// TwinCAT 3 PLC project SlaveController
// ProgramVersion: 3.1.4024.0
// libraries:
//   Tc2_Math, * (Beckhoff Automation GmbH)
//   Tc2_Standard, * (Beckhoff Automation GmbH)
//   Tc2_System, * (Beckhoff Automation GmbH)
//   Tc2_Utilities, * (Beckhoff Automation GmbH)
//   Tc3_Module, * (Beckhoff Automation GmbH)
// project tree:
//   AgiMaths/ deg2rad.TcPOU, sign.TcPOU (not stored), addVec7.TcPOU (not stored), atan2.TcPOU (not stored), cot.TcPOU (not stored)
//   AgiMaths/Frames/ DHTrans.TcPOU (not stored), rotX.TcPOU (not stored), rotY.TcPOU (not stored), rotZ.TcPOU (not stored), transform.TcPOU (not stored)
//   AgiMaths/MatrixLib/ cross.TcPOU (not stored), Det5.TcPOU (not stored), Det6.TcPOU (not stored), Det7.TcPOU (not stored), invMat6.TcPOU, invMat6Old.TcPOU (not stored), invMat3.TcPOU (not stored), invMat7.TcPOU (not stored), Mat3T.TcPOU (not stored), matAdd.TcPOU (not stored), matMultiNum.TcPOU (not stored), matMultiply.TcPOU (not stored), matMultiVec.TcPOU (not stored), matSelfAdd.TcPOU (not stored), matSelfSub.TcPOU (not stored), matSub.TcPOU (not stored), matTranspose.TcPOU (not stored), rot2AngAxis.TcPOU (not stored), vecAdd.TcPOU (not stored), vecNorm.TcPOU (not stored), normVec.TcPOU (not stored), vecSelfMultiNum.TcPOU (not stored), vecMultiNum.TcPOU (not stored), vecSub.TcPOU (not stored)
//   DUTs/Enum/ E_SetupArmState.TcDUT, E_DriverCtrlWord.TcDUT (not stored), E_DriverOPMode.TcDUT (not stored), E_DriverStatusWord.TcDUT (not stored)
//   DUTs/Structure/MasterSlaveCommunication/ E_InstrumentType.TcDUT (not stored), E_MasterArmState.TcDUT (not stored), E_MatchedMasterArmIdx.TcDUT (not stored), E_MatchedSlaveArmIdx.TcDUT (not stored), E_SlaveArmState.TcDUT, ST_InstruStatus.TcDUT (not stored), ST_MasterStatus.TcDUT (not stored), ST_SlaveStatus.TcDUT (not stored)
//   DUTs/Structure/ ST_SetupArmCtrlCmds.TcDUT (not stored), ST_SetupInputDataPool.TcDUT (not stored), ST_SlaveArmCtrlCmds.TcDUT, ST_SlaveInputDataPool.TcDUT, ST_InstruParameters.TcDUT, ST_Frame.TcDUT (not stored)
//   DUTs/Structure/TasksCommunication/ ST_SetupStatus.TcDUT, ST_SetupJointData.TcDUT (not stored), ST_SlaveDynaData.TcDUT (not stored), ST_SlaveUIData.TcDUT, ST_CartStatus.TcDUT (not stored), ST_MasterJointData.TcDUT (not stored), ST_MotorInputs.TcDUT (not stored), ST_MotorOutputs.TcDUT (not stored), ST_SlaveJointData.TcDUT, ST_SafetyData.TcDUT (not stored)
//   DUTs/Type/ Mat34.TcDUT (not stored), Mat37.TcDUT (not stored), Mat43.TcDUT (not stored), Mat4d.TcDUT (not stored), Mat5d.TcDUT (not stored), Mat67.TcDUT (not stored), Mat6d.TcDUT (not stored), Mat76.TcDUT (not stored), Mat7d.TcDUT (not stored), Vec4d.TcDUT (not stored), Vec4i.TcDUT (not stored), Vec5d.TcDUT (not stored), Vec5i.TcDUT (not stored), Vec6i.TcDUT (not stored), Vec8d.TcDUT (not stored), Vec8i.TcDUT (not stored), Mat3d.TcDUT (not stored), Vec3d.TcDUT (not stored), Vec6d.TcDUT (not stored), Vec7d.TcDUT (not stored), Vec7i.TcDUT (not stored)
//   FBs_BasicControllers/ FBGripControl.TcPOU (not stored), FBMacroJntControl.TcPOU, FB_PID.TcPOU (not stored)
//   FBs_RobotDynamics/ FB_SlaveGravity.TcPOU, FB_setupSlaveGravity.TcPOU (not stored)
//   FBs_Robots/ FB_Instrument.TcPOU, FB_SetupArm.TcPOU, FB_SlaveJoint.TcPOU, FB_SetupJoint.TcPOU, FB_SetupRobot.TcPOU, FB_JointBase.TcPOU, FB_SlaveArm.TcPOU, FB_SlaveRobot.TcPOU
//   FBs_SetupControllers/ FB_SetupCtrlManualAdjust.TcPOU (not stored), FB_SetupCtrlHold.TcPOU, FB_SetupArmCtrlBase.TcPOU (not stored), FB_SetupCtrlAutoAdjust.TcPOU (not stored), FB_SetupCtrlCart.TcPOU, FB_SetupCtrlError.TcPOU (not stored), FB_SetupCtrlGraCali.TcPOU, FB_SetupCtrlInit.TcPOU (not stored), FB_SetupCtrlPackage.TcPOU, FB_SetupCtrlSelfCheck.TcPOU, I_SetupArmCtrl.TcIO
//   FBs_SlaveControllers/ FB_SlaveCtrlPackage.TcPOU (not stored), FB_SlaveCtrlEndoscope.TcPOU, FB_SlaveCtrlCart.TcPOU (not stored), FB_SlaveCtrlScopeReady.TcPOU, FB_SlaveCtrlSelfCheck.TcPOU, FB_SlaveCtrlError.TcPOU (not stored), FB_SlaveCtrlInstruReady.TcPOU (not stored), FB_SlaveCtrlMasterSlave.TcPOU, FB_SlaveCtrlMountInstru.TcPOU, FB_SlaveCtrlAdjust.TcPOU, FB_SlaveCtrlMountPanel.TcPOU, FB_SlaveCtrlPanelReady.TcPOU (not stored), FB_SlaveCtrlMountScope.TcPOU (not stored), FB_SlaveCtrlGraCali.TcPOU, FB_SlaveCtrlInit.TcPOU (not stored), FB_SlaveCtrlStandBy.TcPOU, FB_SlaveArmCtrlBase.TcPOU, I_SlaveArmCtrl.TcIO (not stored)
//   FBs_TrajectoryPlanning/ FB_BasicDoubleS.TcPOU (not stored), FB_trajBase.TcPOU (not stored), FB_TrajMoveJ.TcPOU, FB_setupTrajMoveJ.TcPOU, linear_trajectory_with_quintic_polynomial_blends.TcPOU (not stored), quintic_spline_curve.TcPOU (not stored), Quintic_spline_curve_factor.TcPOU (not stored), TrapezoIDal_velocity_trajectory.TcPOU (not stored)
//   FBs_TrajectoryPlanning/OTG/ FB_secOrdTrajFilter.TcPOU (not stored), FB_thirdOrdTrajFilter.TcPOU (not stored)
//   FBs_Filters/ FB_LowPassFilter.TcPOU (not stored)
//   GVLs/ GVL_CartParameters.TcGVL (not stored), GVL_InstruCtrlParams.TcGVL, GVL_MathDefine.TcGVL, GVL_SafetyParameters.TcGVL (not stored), GVL_SystemParameters.TcGVL
//   GVLs/SetupArms/ GVL_SetupJointEncoderCaliData.TcGVL, GVL_SetupMotorParameters.TcGVL, GVL_SetupArmKinematic.TcGVL, GVL_SetupControlParameters.TcGVL (not stored)
//   GVLs/SlaveArms/ GVLs_SlaveArmDynamics.TcGVL, GVLs_SetupSlaveArmDynamics.TcGVL, GVL_SlaveArmKinematic.TcGVL, GVL_SlaveControlParameters.TcGVL, GVL_SlaveMotorParameters.TcGVL, GVL_SlaveJointEncoderCaliData.TcGVL
//   Mains/ SetupArmControl.TcPOU (not stored), SlaveArmControl.TcPOU, RobotDynamics.TcPOU
//   / TaskDynamic.TcTTO (not stored), TaskSetupArmControl.TcTTO, TaskSlaveArmControl.TcTTO
// real-time tasks:
//   TASK TaskSlaveArmControl: cycle T#250us, priority 1, ADS port 350
//   TASK TaskDynamic: cycle T#1ms, priority 2, ADS port 351
//   TASK TaskSetupArmControl: cycle T#1ms, priority 3, ADS port 352

CONFIGURATION SlaveController
    RESOURCE PLC ON TwinCAT3
        TASK TaskSetupArmControl(INTERVAL := T#1ms, PRIORITY := 3);
        TASK TaskSlaveArmControl(INTERVAL := T#250us, PRIORITY := 1);
        PROGRAM SetupArmControl WITH TaskSetupArmControl : SetupArmControl;
        PROGRAM SlaveArmControl WITH TaskSlaveArmControl : SlaveArmControl;
    END_RESOURCE
END_CONFIGURATION

// ---- DUTs/Enum/E_SetupArmState.TcDUT
TYPE E_SetupArmState :
(
	SetupArmState_Error := 1,
	SetupArmState_Init :=2,
	SetupArmState_SelfCheck :=3,
	SetupArmState_Hold :=4,
	SetupArmState_ManulAdjust :=5,
	SetupArmState_AutoAdjust :=6,
	SetupArmState_Package :=7,
	SetupArmState_Cart := 8,
	SetupArmState_GravityCali := 9,
	
	SetupArmState_totalNum :=SetupArmState_GravityCali
);
END_TYPE

// ---- DUTs/Structure/MasterSlaveCommunication/E_SlaveArmState.TcDUT
TYPE E_SlaveArmState :
(
	SlaveArmState_Error := 1,
	SlaveArmState_Init :=2,
	SlaveArmState_SelfCheck :=3,
	SlaveArmState_Standby :=4,
	SlaveArmState_MountPanel:=5,
	SlaveArmState_PanelReady :=6,
	SlaveArmState_MountInstru :=7,
	SlaveArmState_InstruReady :=8,
	SlaveArmState_MasterSlave :=9,
	SlaveArmState_MountScope :=10,
	SlaveArmState_ScopeReady :=11,
	SlaveArmState_EndoScope :=12,
	SlaveArmState_Adjust :=13,	
	SlaveArmState_Package :=14,  		 //包装
	SlaveArmState_Cart := 15,    			 //搬运
	SlaveArmState_GravityCali := 16, 	 //重力标定
	
	SlaveArmState_totalNum :=SlaveArmState_GravityCali
);
END_TYPE

// ---- DUTs/Structure/TasksCommunication/ST_SetupStatus.TcDUT
TYPE ST_SetupStatus :
STRUCT
	// state machine
	m_armState:ARRAY[1..g_sArmNum] OF E_SetupArmState:=[g_sArmNum(SetupArmState_Init)];
	
	// current pose of set arm distal end
	m_curEndPose:ARRAY[1..g_sArmNum] OF ST_Frame;
	
	// position of remote center point
	m_rcPos :ARRAY[1..g_sArmNum] OF Vec3d;
END_STRUCT
END_TYPE

// ---- DUTs/Structure/TasksCommunication/ST_SlaveUIData.TcDUT
// Output from UI controller
// Input to slave arm control task and cart control task  
TYPE ST_SlaveUIData :
STRUCT
	m_slaveArmDisableFlag :Vec4i:=[0, 0, 0, 0];
END_STRUCT
END_TYPE

// ---- DUTs/Structure/TasksCommunication/ST_SlaveJointData.TcDUT
TYPE ST_SlaveJointData :
STRUCT
	
	// joint position compute with motor encoder
	m_curMotorPos :ARRAY[1..g_sArmNum] OF Vec8d;
	
	// joint position compute with link/abs encoder
	m_curLinkPos :ARRAY[1..g_sArmNum] OF Vec8d;
	
	// target joint position 
	m_cmdJntPos :ARRAY[1..g_sArmNum] OF Vec8d;
	
	// current joint position 
	m_curJntPos :ARRAY[1..g_sArmNum] OF Vec8d;
	
	// target joint velocity 
	m_cmdJntVel :ARRAY[1..g_sArmNum] OF Vec8d;
	
	// current joint position 
	m_curJntVel :ARRAY[1..g_sArmNum] OF Vec8d;
	
	// command joint torque 
	m_cmdJntTrq :ARRAY[1..g_sArmNum] OF Vec8d;
	
	// current joint torque 
	m_curJntTrq :ARRAY[1..g_sArmNum] OF Vec8d;
	
	// raw joint current  
	m_rawJntCurrent :ARRAY[1..g_sArmNum] OF Vec8d;
	
	// filtd  joint current  
	m_filtJntCurrent :ARRAY[1..g_sArmNum] OF Vec8d;
	
	// command joint current 
	m_cmdJntCurrent :ARRAY[1..g_sArmNum] OF Vec8d;
END_STRUCT
END_TYPE

// ---- DUTs/Structure/ST_SlaveArmCtrlCmds.TcDUT
TYPE ST_SlaveArmCtrlCmds :
STRUCT
	// arm control data
	m_jntEnableFlag : Vec8i;
	m_jntOPMode : Vec8i;
	m_cmdJntPos : VEC8d;
	m_cmdJntVel : VEC8d;
	m_cmdJntAcc : VEC8d;
	m_cmdJntTrq : VEC8d;
	m_cmdCartPose : ST_Frame;
	m_cmdCartTwist : Vec6d;
	m_ratedCur : VEC8d;
	
END_STRUCT
END_TYPE

// ---- DUTs/Structure/ST_SlaveInputDataPool.TcDUT
// Struct contains all data from other tasks and controller used for slave control
TYPE ST_SlaveInputDataPool :
STRUCT
		
	// UI information, import from UI controller
	m_UIData AT %I*:ST_SlaveUIData;
	
	// safety information, import from safety check task
	m_safetyData AT %I*: ST_SafetyData;
	
	// cart information, import from other task
	m_cartStatus AT %I*:ST_CartStatus;
	
	// master robot information, import from other device
	m_masterStatus AT %I*:ST_MasterStatus;
	
	// setup arms infromation;
	m_setupArmStates AT %i* : ST_SetupArmStatus;
	
	// slave dynamic data
	m_slaveDynaData AT %I* : ST_SlaveDynaData;
	
END_STRUCT
END_TYPE

// ---- DUTs/Structure/ST_InstruParameters.TcDUT
 // instrumetn kinematic paramters
TYPE ST_InstruParameters :
STRUCT	
		
	m_rodLength:LREAL:=0.5392; //器械杆长
	m_headLength:LREAL :=0.01;
	m_fingerLenght:LREAL :=0;//器械头端长度 
	
	kx:lreal:=1;
	ky:lreal:=1;
	kz:lreal:=1;

	k13:LREAL:=0.775;
	k23:LREAL:=0.775;
	m_openAngleDir:INT:=-1;

	Len_fixed_point:LREAL:=0.2;	//不动点距离安装面的长度
	Len_mounting_surface:LREAL:=0.009; //器械安装面距离滑块的长度(图中的L3)
	Len_Hight:lreal:=0; //器械杆的高度
	slope_angle:LREAL:=0; //如果器械是摄像头，还需要考虑摄像头的斜面角度
	open_angle_max:LREAL:=1.57;

END_STRUCT
END_TYPE

// ---- GVLs/GVL_InstruCtrlParams.TcGVL
// TODO： Code review and refined
VAR_GLOBAL
	
	//器械相关
	Head_Len_1:ARRAY[1..30] OF LREAL:=[1,1,1,1,1,1,	0.01950, 0.0096, 0.0109, 0.011,		0.01101, 0.02313, 0.0195, 0.0207, 0.0130, 0.01638, 0.01638, 13(1)	];
	
	camera_slope_angle:LREAL:=30.0*g_deg2Rad;; //摄像头斜面角度
	
	a3:ARRAY[1..30] OF LREAL:=[1,1,1,1,1,1,  0.0089,0.0089,0.010,0.010,		0.0089,0.01065,0.01065,0.01065,0.0089,		0.00935,0.00935,0,0,   4(0), 0.0089, 5(0)];
	k13:ARRAY[1..30] OF LREAL:=[1,1,1,1,1,1, 0.77510204, 0.808510638, 0.62295082, 0.644067797,  0.729166667,  0.5, 0.62295082, 0.62295082,  0.729166667,   -0.734693878,	-0.734693878,    1,      1,   1,	4(1), 0.77510204, 5(1)];
	k23:ARRAY[1..30] OF LREAL:=[1,1,1,1,1,1, 0.77510204, 0.808510638, 0.62295082, 0.644067797,  0.729166667,  0.5, 0.62295082, 0.62295082,  0.729166667,   -0.734693878,	-0.734693878,    1,      1,   1,	4(1), 0.77510204, 5(1)  ];
	kx:ARRAY[1..30] OF LREAL:=[30(-1)];
	ky:ARRAY[1..30] OF LREAL:=[1,1,1,1,1,1,  0.931034483,    0.931034483,      0.931034483,    0.931034483,    0.947368421,    0.931034483,    0.931034483,     0.931034483,     0.931034483,   0.877192982,	0.877192982,    1,      1,   1,	4(1), 0.931034483, 5(1)   ];
	kz:ARRAY[1..30] OF LREAL:=[1,1,1,1,1,1,  0.844827586,    0.810344828,      1.051724138,    1.017241379,    0.842105263,    1.310344828,    1.051724138,     1.051724138,     0.827586207,   0.859649123,	0.859649123,    1,      1,   1,	4(1), 0.844827586, 5(1)  ];
	openAngleDir:ARRAY[1..30] OF INT:=[30(-1)];
	
	rad_30:LREAL:=30.0*g_deg2Rad;  rad_60:LREAL:=60.0*g_deg2Rad;	 rad_38:LREAL:=38.0*g_deg2Rad;	rad_55:LREAL:=55.0*g_deg2Rad;	
	rad_45:LREAL:=45.0*g_deg2Rad; rad_28:LREAL:=28.0*g_deg2Rad; rad_10:LREAL:=10.0*g_deg2Rad;rad_90:LREAL:=90.0*g_deg2Rad;
	open_angle_max:ARRAY[1..30] OF LREAL:=[1,1,1,1,1,1,  rad_45,  rad_30+rad_10,  rad_38+rad_10, rad_38+rad_10,	 rad_30+rad_10, rad_90, rad_45+rad_10, rad_45+rad_10,  rad_60,rad_30,     rad_30,1,1];
	
	tool_name:ARRAY[1..30] OF STRING:=['1','1','1','1','1','1',  'Cadiere Forceps','Large Needle Driver','Mega SutureCut Needle Driver','Large SutureCut Needle Driver',	'RoundTip Scissors','Prograsp',	'Maryland Bipolar Forceps','Fenestrated Bipolar Forceps', 'Monopolar Curved Scissors','Permanent Cautery Hook','Permanent Cautery Spatula','1','1','Camera'];
	
//	Head_Len:ARRAY[1..30] OF LREAL:=[1,1,1,1,1,1,	0.01950, 0.0096, 0.0109, 0.011,		0.01101, 0.02313, 0.0195, 0.0207, 0.0130, 0.01638, 0.01638, 13(1)	];
	Head_Len:ARRAY[1..30] OF LREAL:=[0,0,0,0,0,0,	0, 0.0096, 0.0109,  0.0109,		0, 0, 0, 0, 0, 0, 0, 13(0)	];
		
	//*************************绝对定位精度测试使用*****************************//
	len1:LREAL:=0.5438;  len3:LREAL:=0.009;	len_camera:LREAL:=0.49;//0.477;//0.3035;//0.51	
	Len_Rod:ARRAY[1..30] OF LREAL:=[0,0,0,0,0,  0, len1,len1,len1,len1,	len1,len1,len1,len1,0.54375,	0.5432, 0.5432,0,0,len_camera,     4(0),0.551,5(0)]; //器械的杆长	，ID25号器械是主从延时测试用，长度为533+18
	
	Len_mounting_surface:ARRAY[1..30] OF LREAL:=[0,0,0,0,0,	0,len3,len3,len3,len3,	len3,len3,len3,len3,len3,	len3,len3,0,0,len3,    4(0),len3,5(0)]; //滑块和器械安装面的距离(图中的L3)
	TroCar_Len:LREAL:=0.1;//穿刺器长度、此处使用的是短穿刺器
	Zero_To_Bottom_J8:LREAL:=0.14;//8关节刻度线到最底部长度

	
	// Add by NiFeijian,  new method to mount panel and instrument, can be repalced later
	// joint position of panel locked position
	g_panelLockedPosition :Vec5d:=[0.0, 0.0, 0.0, 0.0, 0.0];	
	
	// motor position when instrument is at zero position
	g_instruZeroPosition :Vec5d :=[0.0, 0.0, 0.0, 0.0, 0.0];// move to instrument chip and read online

END_VAR

// ---- GVLs/GVL_MathDefine.TcGVL
VAR_GLOBAL CONSTANT
	g_smallNum :LREAL := 1E-6;
	g_smallAng :LREAL := 0.01*PI/180;
	g_largeNum: LREAL :=1E16;
	g_deg2Rad :LREAL := pi/180.0;
	g_rad2Deg :LREAL := 180.0/pi;
	
	g_eye3d :Mat3d:=[1, 0, 0,
					 0, 1, 0,
					 0, 0, 1];
	g_eye4d :Mat4d:=[1, 0, 0, 0,
					 0, 1, 0, 0,
					 0, 0, 1, 0,
					 0, 0, 0, 1];
	g_zeorMat3d :Mat3d:=[9(0)];
	
	g_zeroMat6d :Mat6d:=[36(0)];
	g_zeroMat7d :Mat7d:=[49(0)];
	g_eye7d :Mat7d:=[1, 0, 0, 0, 0, 0, 0, 
					 0, 1, 0, 0, 0, 0, 0, 
					 0, 0, 1, 0, 0, 0, 0, 
					 0, 0, 0, 1, 0, 0, 0,
					 0, 0, 0, 0, 1, 0, 0,
					 0, 0, 0, 0, 0, 1, 0,
					 0, 0, 0, 0, 0, 0, 1];
	
	g_zeroVec3d :Vec3d:= [3(0)];
	g_onesVec3d: Vec3d:=[3(1)];
	
	g_zeroVec6d: Vec6d:=[6(0)];
	g_onesVec6d: Vec6d:=[6(1)];
	
	g_zeroVec5d: Vec5d:=[5(0)];
	g_onesVec5d: Vec5d:=[5(1.0)];
	g_zeroVec5i: Vec5i:=[5(0)];
	g_onesVec5i: Vec5i:=[5(1)];
	
	g_zeroVec7d: Vec7d:=[7(0)];
	g_onesVec7d: Vec7d:=[7(1.0)];
	g_zeroVec7i: Vec7i:=[7(0)];
	g_onesVec7i: Vec7i:=[7(1)];
	g_zeroVec8d: Vec8d:=[8(0)];
	g_onesVec8d: Vec8d:=[8(1.0)];
	g_zeroVec8i: Vec8i:=[8(0)];
	g_onesVec8i: Vec8i:=[8(1)];
	
	g_setupAllPosMode:Vec5i:=[5(DriverOPMode_Pos)];
	g_setupAllTrqMode:Vec5i:=[5(DriverOPMode_Trq)];
	g_slaveAllPosMode:Vec8i:=[8(DriverOPMode_Pos)];
	g_slaveAllTrqMode:Vec8i:=[8(DriverOPMode_Trq)];
	g_slaveAllPosTrqMode:Vec8i:=[8(DriverOPMode_PosTrq)];
	
	
END_VAR

// ---- GVLs/GVL_SystemParameters.TcGVL
VAR_GLOBAL CONSTANT
	
	g_mArmNum :INT := 2;	
	g_mJntNum :INT := 7;	
	g_sArmNum :INT := 4;	
	g_sJntNum :INT := 8;
	g_setupJntNum :INT :=5;
	g_cartDofs :INT :=6;
	
	
	
	// control loop interval for each task
	g_slaveArmCtrlCycleTime :LREAL :=0.00025;
	g_slaveArmCtrlFreq :LREAL :=1.0/g_slaveArmCtrlCycleTime;
	g_armDynamicCycleTime :LREAL := 0.001;
	g_armDynamicFreq :LREAL := 1.0/g_armDynamicCycleTime;
	g_setupArmCtrlCycleTime :LREAL := 0.001;
	g_setupArmCtrlFreq :LREAL := 1.0/g_setupArmCtrlCycleTime;
	g_cartCtrlCycleTime :LREAL := 0.001;
	g_cartCtrlFreq :LREAL := 1.0/g_cartCtrlCycleTime;
	
	// wait time before robot init  for ethercat to stablize 
	g_robotInitWaitTime : LREAL := 1.0;

END_VAR

// ---- GVLs/SetupArms/GVL_SetupJointEncoderCaliData.TcGVL
{attribute 'qualified_only'}
VAR_GLOBAL
		// abolute encoder expanded limit buffer in case there is calibrtion error at limit position
	g_linkEncLimitBuffer : DINT := 5000;
	
	// absolute encoder value at minimal joint positon
	g_minLinkEncoder :ARRAY[1..g_sArmNum, 1..g_setupJntNum] OF DINT :=
		[0, 0, 0, 0, 0,
		 0, 0, 0, 0, 0,
		 0, 0, 0, 0, 0,
		 0, 0, 0, 0, 0];
		 
	// absolute encoder value at maximum joint positon
	g_maxLinkEncoder :ARRAY[1..g_sArmNum, 1..g_setupJntNum] OF DINT :=
		[0, 0, 0, 0, 0,
		 0, 0, 0, 0, 0,
		 0, 0, 0, 0, 0,
		 0, 0, 0, 0, 0];
	
	// absolute encoder value at calibrated positon
	g_caliLinkEncoder :ARRAY[1..g_sArmNum, 1..g_setupJntNum] OF DINT :=
		[0, 0, 0, 0, 0,
		 0, 0, 0, 0, 0,
		 0, 0, 0, 0, 0,
		 0, 0, 0, 0, 0];
	
	 // if absolute encoder value cross zeros within joint motion range
	g_linkEncZeroCross :ARRAY[1..g_sArmNum, 1..g_setupJntNum] OF INT :=
		[0, 0, 0, 0, 0,
		 0, 0, 0, 0, 0,
		 0, 0, 0, 0, 0,
		 0, 0, 0, 0, 0];
	
	// flag if joint can rotate multiple cycles
	g_multipleCyclesJoint :ARRAY[1..g_sArmNum, 1..g_setupJntNum] OF INT :=
		[0, 0, 0, 0, 0,
		 0, 0, 0, 0, 0,
		 0, 0, 0, 0, 0,
		 0, 0, 0, 0, 0];
		 
	// joint position at link encoder calibrated point
	g_linkEncCaliJntPos :ARRAY[1..g_setupJntNum] OF LREAL :=
		[0.0, 0.0, 0.0, 0.0, 0.0];
		
END_VAR

// ---- GVLs/SetupArms/GVL_SetupMotorParameters.TcGVL
{attribute 'global_init_slot' := '49991'}
{attribute 'qualified_only'}
VAR_GLOBAL CONSTANT
	// encoder resolution
	g_incEncoderRes :ARRAY[1..g_setupJntNum] OF DINT :=[5(65536)];
	g_absEncoderRes :ARRAY[1..g_setupJntNum] OF DINT :=[16777216,8192, 8192, 2(16777216)];
	
	// reduction ratio
	g_motorReduction :ARRAY[1..g_setupJntNum] OF LREAL :=[1,1,2*pi/0.020,81,161];
	g_absEncoderReduction :ARRAY[1..g_setupJntNum] OF LREAL :=[1.0, 0.002/(2*pi) , 0.002/(2*PI), 1.0, 1.0];
	
	// motor parameters
	g_motorTrqConst :ARRAY[1..g_setupJntNum] OF LREAL :=[ 1,1,0.16,0.1,0.16];
	g_motorMaxCurrent :ARRAY[1..g_setupJntNum] OF LREAL :=[ 1,1,5600,3800,5600];//mA
	
	// motor and absEncoder direction
	g_motorDir :ARRAY[1..g_setupJntNum] OF INT :=[-1, -1, 1, -1, 1];
														
	g_asbEncoderDir :ARRAY[1..g_setupJntNum] OF INT :=[1, 1, -1, -1, -1];
													
																 
	// joint position limit
	g_minJntPos: ARRAY[1..g_setupJntNum] OF LREAL:=[-1,	-1,	-1, -1, -1];	
	g_maxJntPos: ARRAY[1..g_setupJntNum] OF LREAL:=[1, 1, 1, 1, 1];	
	
	// joint velocity limit
	g_maxJntVel :ARRAY[1..g_setupJntNum] OF LREAL :=[0.1, 0.1, 0.1, 0.1, 0.1];
	
END_VAR

// ---- GVLs/SetupArms/GVL_SetupArmKinematic.TcGVL
// use slot attribute larger than 49990, which is the default one, if it depends on variable in other file
{attribute 'global_init_slot' := '49991'} 
{attribute 'qualified_only'}
VAR_GLOBAL CONSTANT 

(* 
% paramters definiton:
% d1: distance from joint1 to remote center
% L: instrument length
% a: distance from joint5 to joint 6 on tool
% b: distantce form joint 6 to tcp on tool
% DH definition:
% index    alpha   a   theta   d
% 1        90      0   q1      d1
% 2        -90     0   q2      0
% 3        -90     0   0       q3
% 4        0       0   q4      -L
% 5        90      0   q5      0
% 6        90      a   q6      0
% tcp      0       b   0       0


g_d1:LREAL:=0.8046229;
g_L :LREAL:= 0.3;// need to be replace by real instrument parameters;
g_a : LREAL :=0.01;// need to be replace by real instrument parameters;
g_b :LREAL :=0;// need to be replace by real instrument parameters;

//alpha,a,d,theta	
g_slaveArmDH:ARRAY[1..9,1..4] OF LREAL :=[PI/2,	0,		g_d1,	0,      
											-pi/2,	0,		0,		0,
											-PI/2,	0,		0,		0,
									        0,		0,		-g_L,	0,       
											pi/2,	0,		0,		0,
								            pi/2,	g_a,	0,		0,
							         		0,		g_b, 	0,		0];

*)
END_VAR

// ---- GVLs/SlaveArms/GVLs_SlaveArmDynamics.TcGVL
{attribute 'global_init_slot' := '49992'}
VAR_GLOBAL CONSTANT
	
(*graParam=[ 9.8*mx0,...
           9.8*m5,...
           0.41601*m2 + 0.41601*m3 + 0.0000216012*m4 + 0.0000216012*m5 + 9.8*mx1 - 1.3639*mx3 - 9.70463*my3,...
           4.92539*m1 + 4.92539*m2 + 4.92539*m3 + 7.8853*m4 + 7.8853*m5 + 9.70463*mx3 - 9.8*my0 - 1.3639*my3 + 9.8*mz1,...
           9.8*mz2 - 9.8*my5 - 9.8*my1 + 9.8*mz3 + 9.8*mz4,...
           2.19651*m3 + 2.19651*m4 + 0.00000258969*m5 + 8.64766*mx2 - 4.61063*my2 + 9.8*my4 + 9.8*mz5,...
           1.1711*m3 + 1.1711*m4 + 0.00000122416*m5 + 4.61063*mx2 - 9.8*mx4 - 9.8*mx5 + 8.64766*my2]';
*)
				
	// robot No.4
	g_gravityParam :ARRAY[1..4,1..5] OF REAL := 
	[-0.5414,    1.2050,    0.4391,    0.4801,    0.6717,
	 -0.3477,    1.1457,    0.4601,    0.4529,    0.7010,
	 -0.3373,    1.1255,    0.4497,    0.4801,    0.6666,
	 -0.3639,    1.2385,    0.5290,    0.4801,    0.6862];
	 
	g_gravityTrocar :ARRAY[1..5] OF REAL :=[-0.0063,    0.0113,   -0.0026,   -0.0149,    0.0021];
	g_gravityInstrument :ARRAY[1..5] OF REAL :=[-0.0082,   -0.0347,   -0.0132,   -0.0044,    0.3037];
	g_gravityEndoscope :ARRAY[1..5] OF REAL :=[ -0.1037,   -0.0120,    0.0441,    0.0183,    1.0935];
	

END_VAR

// ---- GVLs/SlaveArms/GVLs_SetupSlaveArmDynamics.TcGVL
{attribute 'global_init_slot' := '49992'}
{attribute 'qualified_only'}
VAR_GLOBAL CONSTANT
	
(*graParam=[ mz2 - my5 - my1 + mz3 + mz4,...
			   0.22413*m3 + 0.22413*m4 + 2.6425e-7*m5 + 0.88241*mx2 - 0.47047*my2 + 1.0*my4 + 1.0*mz5,...
			   0.1195*m3 + 0.1195*m4 + 1.2491e-7*m5 + 0.47047*mx2 - mx4 - mx5 + 0.88241*my2,...
			  0.04245*m2 + 0.04245*m3 + 2.2042e-6*m4 + 2.2042e-6*m5 + 1.0*mx1 - 0.13917*mx3 - 0.99027*my3,...
			  m5]'
*)
				
	// robot No.4
	g_gravityParam :ARRAY[1..4,1..7] OF REAL := 
	[-0.5414,    1.2050,    0.4391,    0.4801,    0.6717,
	 -0.3477,    1.1457,    0.4601,    0.4529,    0.7010,
	 -0.3373,    1.1255,    0.4497,    0.4801,    0.6666,
	 -0.3639,    1.2385,    0.5290,    0.4801,    0.6862];
	 
	g_gravityTrocar :ARRAY[1..7] OF REAL :=[-0.0063,    0.0113,   -0.0026,   -0.0149,    0.0021];
	g_gravityInstrument :ARRAY[1..7] OF REAL :=[-0.0082,   -0.0347,   -0.0132,   -0.0044,    0.3037];
	g_gravityEndoscope :ARRAY[1..7] OF REAL :=[ -0.1037,   -0.0120,    0.0441,    0.0183,    1.0935];
	
(*	// link mass [m1, m2, m3, m4, m5, m6, m7, m8, m9]
	g_linkMass :ARRAY[1..9] OF LREAL :=[2.676, 0.825, 0.547, 0.25, 0.195, 0.194, 0.05, 0.111, 0.09] ;
	
	// lin center of amss
	g_linkCOM :ARRAY[1..9,1..3] OF LREAL := [   1.376E-3,    -1.019E-3,  -81.464E-3,
										   90.622E-3,   -0.113E-3,  15.088E-3,
										   167.4E-3,    3.7E-3,     -0.438E-3,
										   0.1E-3,      98.49E-3,   -55.74E-3,
										   0.12E-3,     76.667E-3,  -36E-3,
										   0,           -61.63E-3,  27.3E-3,
										   0.06E-3,     -0.08E-3,   17.671E-3,
										   11E-3,       -3.364E-3,  39.265E-3,
										   143e-3,      0.495e-3,   24.253e-3];
	// link  inertial
    // [Ixx,Iyy,Izz, Ixy,Ixz, Iyz]
 	g_linkInertia :ARRAY[1..9,1..6] OF LREAL :=[  19.63E-3,   16.43E-3,  12.7E-3,   -0.3222E-3,    -0.667E-3,     -0.0268E-3,
												   1.017E-3,   6.637E-3,  5.935E-3,  -0.037E-3,     -0.238E-3,     0.06E-3,
												   0.161E-3,   9.572E-3,  9.586E-3,  0.0447E-3,     0.0277E-3,     0.465E-6,
												   0.992E-3,   0.707E-3,  0.335E-3,  0.2E-6,     2E-6,       0.224E-3,
												   0.402E-3,   0.25E-3,   0.186E-3,  0.002E-6,   -1.2E-6,    0.106E-3,
												   0.281E-3,   0.178E-3,  0.137E-3,  0.076E-6,   0.09E-6,    0.056E-3,
												   0.0255E-3,  0.0259E-3, 5.96E-6,0.34E-6,    -3E-9,      24E-9,
												   0.033E-3,   0.0976E-3, 0.126E-3,  3E-6,       -5E-6,      -0.162E-6,
												   4.9E-6,  0.757E-3,  0.760E-3,  2.6E-6,     -5.3E-6,    -18E-9];


	//  motor inertial at link size
	g_motorInertia :ARRAY[1..7] OF LREAL := [34.7E-7, 34.7E-7, 34.7E-7, 9.26E-7, 0.495E-7, 0.495E-7, 0.495E-7];
	*)
END_VAR

// ---- GVLs/SlaveArms/GVL_SlaveArmKinematic.TcGVL
// use slot attribute larger than 49990, which is the default one, if it depends on variable in other file
{attribute 'global_init_slot' := '49991'} 
{attribute 'qualified_only'}
VAR_GLOBAL CONSTANT 

(* 
% paramters definiton:
% d1: distance from joint1 to remote center
% L: instrument length
% a: distance from joint5 to joint 6 on tool
% b: distantce form joint 6 to tcp on tool
% DH definition:
% index    alpha   a   theta   d
% 1        90      0   q1      d1
% 2        -90     0   q2      0
% 3        -90     0   0       q3
% 4        0       0   q4      -L
% 5        90      0   q5      0
% 6        90      a   q6      0
% tcp      0       b   0       0

*)
g_d1:LREAL:=0.8046229;
g_L :LREAL:= 0.3;// need to be replace by real instrument parameters;
g_a : LREAL :=0.01;// need to be replace by real instrument parameters;
g_b :LREAL :=0;// need to be replace by real instrument parameters;

//alpha,a,d,theta	
g_masterArmDH:ARRAY[1..9,1..4] OF LREAL :=[PI/2,	0,		g_d1,	0,      
											-pi/2,	0,		0,		0,
											-PI/2,	0,		0,		0,
									        0,		0,		-g_L,	0,       
											pi/2,	0,		0,		0,
								            pi/2,	g_a,	0,		0,
							         		0,		g_b, 	0,		0];


END_VAR

// ---- GVLs/SlaveArms/GVL_SlaveControlParameters.TcGVL
{attribute 'global_init_slot' := '49991'}
{attribute 'qualified_only'}
VAR_GLOBAL CONSTANT
	// master arm joint position controller parameters
	g_posKp :ARRAY[1..g_sJntNum] OF LREAL :=[2000.0, 2000.0, 18000.0, 35.0, 35.0, 35.0, 35.0, 0];
	g_posKd :ARRAY[1..g_sJntNum] OF LREAL :=[200.0, 200.0, 200.0, 2.0, 2.0, 2.0, 2.0, 0];
	g_posKi :ARRAY[1..g_sJntNum] OF LREAL :=[20000.0, 20000.0, 30000.0, 100.0, 100.0, 100.0, 100.0,0];
	g_posKiLimit :ARRAY[1..g_sJntNum] OF LREAL :=[2500,2500,  250, 5(200)];// define in current
	g_posCtrlLimit :ARRAY[1..g_sJntNum] OF LREAL :=[5600,5600,  500, 5(500)];// define in current
	
	// control tolerance
	g_jntCtrlPosTol :LREAL :=0.2*g_deg2Rad;
	g_cartCtrlPosTol :LREAL :=0.0002;
	g_cartCtrlOriTol :LREAL :=0.2*g_deg2Rad;
	
	// filter cut-off frequency for velocity and torque
	g_curJntVelLpfCutoffFreq :LREAL := 30;
	g_cmdJntPosLpfCutoffFreq :LREAL := 30;
	g_cmdJntTrqLpfCutoffFreq :LREAL := 300;
	g_curJntTrqLpfCutoffFreq :LREAL := 300;
	
	// controller would keep command unchanged when error 
	// between command and current value is less than this value
	g_jntCtrlErrForCmdHold :LREAL :=1.0*g_deg2Rad;
	
	// joint is assumed to be static if velocity is less than this value
	g_jntStaticVelThres :LREAL :=0.2*g_deg2Rad;
	
	// slave self-check motion parameters
	g_selfCheckMotionNum :INT :=2;
	g_selfCheckPosture:ARRAY [1..g_selfCheckMotionNum, 1..g_sJntNum] OF LREAL:=[PI/4, -PI/4, 0.25, pi, pi, pi, pi, pi, 
							 			  			0.0, 	-PI/2, 0.4, 	0, 0, 0, 0,0];
	g_selfCheckMaxjntVel:Vec8d:=[0.2, 0.2, 0.1, 5(1.0)];
	g_selfCheckMaxjntAcc:Vec8d:=[1.0, 1.0, 0.5, 5(2.0)];
	g_selfCheckMaxjntJerk:Vec8d:=[2.0,2.0, 1.0, 5(4.0)];
	
END_VAR

// ---- GVLs/SlaveArms/GVL_SlaveMotorParameters.TcGVL
{attribute 'global_init_slot' := '49991'}
{attribute 'qualified_only'}
VAR_GLOBAL CONSTANT
	// encoder resolution
	g_incEncoderRes :ARRAY[1..g_sJntNum] OF DINT :=[8(65536)];
	g_absEncoderRes :ARRAY[1..g_sJntNum] OF DINT :=[8(16777216)];
	
	// reduction ratio
	g_motorReduction :ARRAY[1..g_sJntNum] OF LREAL :=[ 81,81,  (66.0/10)*2*pi/0.010, 5(388125.0/4693)];
	g_absEncoderReduction :ARRAY[1..g_sJntNum] OF LREAL :=[2(1.0), 2*PI/0.64, 5(1.0)];
	
	// motor parameters
	g_motorTrqConst :ARRAY[1..g_sJntNum] OF LREAL :=[ 0.16,0.16, 0.017,5(0.0193)];
	g_motorMaxCurrent :ARRAY[1..g_sJntNum] OF LREAL :=[ 5600,5600,  500, 5(500)];//mA
	
	// motor encoder direction
	g_motorDir :ARRAY[1..g_sJntNum] OF INT :=[-1, 1, -1, 1, 1, 1, 1, 1];
																 
	// joint position limit
	g_minJntPos: ARRAY[1..g_sJntNum] OF LREAL:=[-pi,	-pi/2,	0.15, 	5(-99*pi)];	
	g_maxJntPos: ARRAY[1..g_sJntNum] OF LREAL:=[pi,	1.196, 	0.58, 		5(99*pi)];
	
	// joint velocity limit
	g_maxJntVel :ARRAY[1..g_sJntNum] OF LREAL :=[1.2, 1.2, 0.2, 5(2*pi)];
	
	// joint SDO address
	g_slaveArmNetID: ARRAY[1..4] OF T_AmsNetId:=['169.254.240.177.5.1','169.254.223.239.7.1','169.254.223.239.9.1','169.254.223.239.10.1'];
	g_slaveJointNetPort:ARRAY[1..g_sArmNum,1..g_sJntNum] OF UINT :=[
		1004,	1005,	1006,	2(1007),	3(1008),
		1006,	1007,	1008,	2(1009),	3(1010),
		1006,	1007,	1008,	2(1009),	3(1010),
		1006,	1007,	1008,	2(1009),	3(1010)];
		
END_VAR

// ---- GVLs/SlaveArms/GVL_SlaveJointEncoderCaliData.TcGVL
{attribute 'qualified_only'}
VAR_GLOBAL CONSTANT
	// abolute encoder expanded limit buffer in case there is calibrtion error at limit position
	g_linkEncLimitBuffer : DINT := 5000;
	
	// absolute encoder value at minimal joint positon
	g_minLinkEncoder :ARRAY[1..g_sArmNum, 1..g_sJntNum] OF DINT :=
		[0, 0, 0, 0, 0, 0, 0, 0,
		 0, 0, 0, 0, 0, 0, 0, 0,
		 0, 0, 0, 0, 0, 0, 0, 0,
		 0, 0, 0, 0, 0, 0, 0, 0];
		 
	// absolute encoder value at maximum joint positon
	g_maxLinkEncoder :ARRAY[1..g_sArmNum, 1..g_sJntNum] OF DINT :=
		[0, 0, 0, 0, 0, 0, 0, 0,
		 0, 0, 0, 0, 0, 0, 0, 0,
		 0, 0, 0, 0, 0, 0, 0, 0,
		 0, 0, 0, 0, 0, 0, 0, 0];
	
	// absolute encoder value at calibrated positon
	g_caliLinkEncoder :ARRAY[1..g_sArmNum, 1..g_sJntNum] OF DINT :=
		[0, 0, 0, 0, 0, 0, 0, 0,
		 0, 0, 0, 0, 0, 0, 0, 0,
		 0, 0, 0, 0, 0, 0, 0, 0,
		 0, 0, 0, 0, 0, 0, 0, 0];
	
	 // if absolute encoder value cross zeros within joint motion range
	 // NOTICE: joint 7 is always 0.
	g_linkEncZeroCross :ARRAY[1..g_sArmNum, 1..g_sJntNum] OF INT :=
		[0, 0, 0, 0, 0, 0, 0, 0,
		 0, 0, 0, 0, 0, 0, 0, 0,
		 0, 0, 0, 0, 0, 0, 0, 0,
		 0, 0, 0, 0, 0, 0, 0, 0];
	
	// flag if joint can rotate multiple cycles
	g_multipleCyclesJoint :ARRAY[1..g_sArmNum, 1..g_sJntNum] OF INT :=
		[0, 0, 0, 1, 1, 1, 1, 1,
		 0, 0, 0, 1, 1, 1, 1, 1,
		 0, 0, 0, 1, 1, 1, 1, 1,
		 0, 0, 0, 1, 1, 1, 1, 1];
		 
	// joint position at link encoder calibrated point
	g_linkEncCaliJntPos :ARRAY[1..g_sJntNum] OF LREAL :=
		[0.0, -PI/2, 0.581633, 5(0.0)];

END_VAR

// ---- FBs_SetupControllers/I_SetupArmCtrl.TcIO
INTERFACE I_SetupArmCtrl

METHOD init : BOOL
VAR_IN_OUT CONSTANT
	i_setupArm	:FB_SetupArm;
END_VAR
VAR_IN_OUT 
	r_setupArmCtrlCmd :ST_SetupArmCtrlCmds;
END_VAR
END_METHOD

PROPERTY isFinished : bool
GET
END_GET
END_PROPERTY

METHOD reset : BOOL
VAR_INPUT
END_VAR
END_METHOD

METHOD run : BOOL
VAR_IN_OUT CONSTANT
	i_setupArm	:FB_SetupArm;
END_VAR
VAR_IN_OUT 
	r_setupArmCtrlCmd :ST_SetupArmCtrlCmds;
END_VAR
END_METHOD

END_INTERFACE

// ---- Mains/SlaveArmControl.TcPOU
PROGRAM SlaveArmControl
VAR
	// flag to init robot
	m_robotInit :BOOL :=FALSE;
	
	// wait time before robot init  for ethercat to be statble 
	m_robotInitWaitTime : LREAL:=0;
	
	// slave robot
	m_slaveRobot:FB_SlaveRobot;
	
	// slave robot information, including arm status and cartesian data
	m_slaveStatus AT %Q* :ST_slaveStatus;
	
	// slave robot joint data
	m_slaveJointsData AT %Q* :ST_slaveJointData;
	
	// all data from other tasks and controller 
	m_slaveInputDataPool : ST_SlaveInputDataPool;

	// code execute time measure
	m_codeTime : Profiler;
	
END_VAR

//m_codeTime(START:=TRUE, RESET:=TRUE);

// wait communication to be stable
IF(m_robotInitWaitTime<g_robotInitWaitTime) THEN
	m_robotInitWaitTime := m_robotInitWaitTime+g_slaveArmCtrlCycleTime;
	RETURN;
END_IF

// robot init
IF m_robotInit =FALSE THEN
	m_slaveRobot.Init();
	m_robotInit:=TRUE;
END_IF

// robot run
m_slaveRobot.run(m_slaveInputDataPool);

// update data pool
m_slaveRobot.getStatus(m_slaveStatus,m_slaveJointsData);

//m_codeTime(START:=FALSE,RESET:=FALSE);

END_PROGRAM

// ---- FBs_Robots/FB_SlaveRobot.TcPOU
FUNCTION_BLOCK FB_SlaveRobot
VAR_INPUT
END_VAR
VAR_OUTPUT
END_VAR
VAR
	// master-slave motion scale
	m_motionScale :LREAL;
	
	// slave arms, responsible for arm kinematic and control
	m_slaveArms :ARRAY[1..g_sArmNum] OF FB_SlaveArm;
	
	// arm state
	m_slaveArmState:ARRAY[1..g_sArmNum] OF E_slaveArmState:=[4(E_SlaveArmState.SlaveArmState_Init)];
	m_lastSlaveArmState:ARRAY[1..g_sArmNum] OF E_slaveArmState:=[4(E_SlaveArmState.SlaveArmState_Init)];
	m_nextSlaveArmState:ARRAY[1..g_sArmNum] OF E_masterArmState:=[4(E_SlaveArmState.SlaveArmState_Init)];
	
	// index(1 to 4) of slave arm which is tele-linked to master arm
	m_teleMasterArmIdx:ARRAY[1..g_sArmNum] OF E_MatchedMasterArmIdx:=[4(MatchedMasterArmIdx_NULL)];
	
	// all arm controller instance 
	m_armCtrlFactory :ARRAY[1..g_sArmNum,1..SlaveArmState_totalNum] OF I_SlaveArmCtrl;
	m_armError :ARRAY[1..g_sArmNum] OF FB_SlaveCtrlError;
	m_armInit :ARRAY[1..g_sArmNum] OF FB_SlaveCtrlInit;
	m_armSelfCheck :ARRAY[1..g_sArmNum] OF FB_SlaveCtrlSelfCheck;
	m_armStandBy :ARRAY[1..g_sArmNum] OF FB_SlaveCtrlStandBy;
	m_mountPanel :ARRAY[1..g_sArmNum] OF FB_SlaveCtrlMountPanel;
	m_panelReady :ARRAY[1..g_sArmNum] OF FB_SlaveCtrlPanelReady;
	m_mountInstru :ARRAY[1..g_sArmNum] OF FB_SlaveCtrlMountInstru;
	m_instruReady :ARRAY[1..g_sArmNum] OF FB_SlaveCtrlInstruReady;
	m_armMasterSlave :ARRAY[1..g_sArmNum] OF FB_SlaveCtrlMasterSlave;
	m_mountScope :ARRAY[1..g_sArmNum] OF FB_SlaveCtrlMountScope;
	m_scopeReady :ARRAY[1..g_sArmNum] OF FB_SlaveCtrlScopeReady;
	m_armEndoscope :ARRAY[1..g_sArmNum] OF FB_SlaveCtrlEndoscope;
	m_armAdjust :ARRAY[1..g_sArmNum] OF FB_SlaveCtrlAdjust;
	m_armPackage :ARRAY[1..g_sArmNum] OF FB_SlaveCtrlPackage;
	m_armCart :ARRAY[1..g_sArmNum] OF FB_SlaveCtrlCart;
	m_armGraCali :ARRAY[1..g_sArmNum] OF FB_SlaveCtrlGraCali;
	
	// arm controller interface
	m_armCtrl :ARRAY[1..g_sArmNum] OF I_SlaveArmCtrl;
	m_armCtrlCmds :ARRAY[1..g_sArmNum] OF ST_SlaveArmCtrlCmds;

END_VAR

METHOD checkTeleMasterArmIdx : BOOL
VAR_INPUT
END_VAR
// TODO: decide the matched master arm index for each slave arm
END_METHOD

METHOD PUBLIC getStatus : BOOL
VAR_IN_OUT
	// slave robot information, including arm status and cartesian data
	r_slaveStatus :ST_SlaveStatus;
	
	// slave robot joint data
	r_slaveJointsData :ST_SlaveJointData;
	
END_VAR

VAR
	i:INT;
END_VAR
r_slaveStatus.m_armState:=m_slaveArmState;
r_slaveStatus.m_teleMasterArmIdx := m_teleMasterArmIdx;

// TODO: project cartesion data to monitor coordinate
FOR i:=1 TO g_sArmNum DO
	
	// instrument data
	r_slaveStatus.m_instruStauts[i].m_type:=m_slaveArms[i].instrument.instruType;
	r_slaveStatus.m_instruStauts[i].m_ready:=m_slaveArms[i].instruOn;
	r_slaveStatus.m_instruStauts[i].m_fingerAngle:=m_slaveArms[i].gripAngle;
	
	// cartesion
	r_slaveStatus.m_curArmPose[i]:=m_slaveArms[i].curCartPose;
	r_slaveStatus.m_curArmTwist[i]:=m_slaveArms[i].curCartTwist;
	// joint
	r_slaveJointsData.m_curMotorPos[i]:=m_slaveArms[i].curMotorPos;
	r_slaveJointsData.m_curLinkPos[i]:=m_slaveArms[i].curLinkPos;
	r_slaveJointsData.m_curJntPos[i]:=m_slaveArms[i].curJntPos;
	r_slaveJointsData.m_curJntVel[i]:=m_slaveArms[i].curJntVel;
	r_slaveJointsData.m_curJntTrq[i]:=m_slaveArms[i].curJntTrq;
	
	// command info
	// cartesion
	r_slaveStatus.m_cmdArmPose[i]:=m_armCtrlCmds[i].m_cmdCartPose;
	r_slaveStatus.m_cmdArmTwist[i]:=m_armCtrlCmds[i].m_cmdCartTwist;
	// joint info
	r_slaveJointsData.m_cmdJntPos[i]:=m_armCtrlCmds[i].m_cmdJntPos;
	r_slaveJointsData.m_cmdJntVel[i]:=m_armCtrlCmds[i].m_cmdJntVel;
	r_slaveJointsData.m_cmdJntTrq[i]:=m_armCtrlCmds[i].m_cmdJntTrq;
	
END_FOR
END_METHOD

METHOD PUBLIC Init : BOOL
VAR_INPUT
END_VAR
VAR
	i:INT;
END_VAR
FOR i:=1 TO g_sArmNum DO
	// arm init
	m_slaveArms[i].Init(i);
	m_slaveArmState[i]:=SlaveArmState_Init;
	m_lastSlaveArmState[i]:=SlaveArmState_Init;
	m_nextSlaveArmState[i]:=SlaveArmState_Init;
	m_teleMasterArmIdx[i]:=MatchedMasterArmIdx_NULL;
	
	// command init
	m_armCtrlCmds[i].m_jntEnableFlag := g_zeroVec8i;
	m_armCtrlCmds[i].m_jntOPMode := g_slaveAllPosMode;
	m_armCtrlCmds[i].m_cmdCartPose := m_slaveArms[i].curCartPose;
	m_armCtrlCmds[i].m_cmdCartTwist := g_zeroVec6d;
	m_armCtrlCmds[i].m_cmdJntPos := m_slaveArms[i].curJntPos;
	m_armCtrlCmds[i].m_cmdJntVel := g_zeroVec8d;
	m_armCtrlCmds[i].m_cmdJntAcc := g_zeroVec8d;
	m_armCtrlCmds[i].m_cmdJntTrq := g_zeroVec8d;
	
	// generate controller factory
	m_armCtrlFactory[i,SlaveArmState_Error] := m_armError[i];
	m_armCtrlFactory[i,SlaveArmState_Init] := m_armInit[i];
	m_armCtrlFactory[i,SlaveArmState_SelfCheck] := m_armSelfCheck[i];
	m_armCtrlFactory[i,SlaveArmState_Standby] := m_armStandBy[i];
	m_armCtrlFactory[i,SlaveArmState_MountPanel] := m_mountPanel[i];
	m_armCtrlFactory[i,SlaveArmState_PanelReady] := m_panelReady[i];
	m_armCtrlFactory[i,SlaveArmState_MountInstru] := m_mountInstru[i];
	m_armCtrlFactory[i,SlaveArmState_InstruReady] := m_instruReady[i];
	m_armCtrlFactory[i,SlaveArmState_MasterSlave] := m_armMasterSlave[i];
	m_armCtrlFactory[i,SlaveArmState_MountScope] := m_mountScope[i];
	m_armCtrlFactory[i,SlaveArmState_ScopeReady] := m_scopeReady[i];
	m_armCtrlFactory[i,SlaveArmState_EndoScope] := m_armEndoscope[i];
	m_armCtrlFactory[i,SlaveArmState_Adjust] := m_armAdjust[i];
	m_armCtrlFactory[i,SlaveArmState_Package] := m_armPackage[i];
	m_armCtrlFactory[i,SlaveArmState_Cart] := m_armCart[i];
	m_armCtrlFactory[i,SlaveArmState_GravityCali] := m_armGraCali[i];
	
	// assign controller
	m_armCtrl[i]:=m_armCtrlFactory[i,m_slaveArmState[i]];
	m_armCtrl[i].Init(m_slaveArms[i],m_armCtrlCmds[i]);
END_FOR
END_METHOD

METHOD PUBLIC run : BOOL
VAR_IN_OUT CONSTANT
	i_slaveInputDataPool:ST_SlaveInputDataPool;
END_VAR
VAR
	i:INT;
END_VAR
m_motionScale := i_slaveInputDataPool.m_masterStatus.m_motionScale;

// state machine transition
stateMachine(i_slaveInputDataPool);

FOR i:=1 TO g_sArmNum DO
	// update dynamic data
	m_slaveArms[i].updateDyna(i_slaveInputDataPool.m_slaveDynaData);
								
	// update slave arm kinematics
	m_slaveArms[i].updateStatus();
	
	// null ptr check
	IF 0 = m_armCtrl[i] THEN
		EXIT;
	END_IF
	
	// run controller
	m_armCtrl[i].run(m_motionScale, m_teleMasterArmIdx[i], m_SlaveArms[i],
						i_slaveInputDataPool.m_MasterStatus,m_armCtrlCmds[i]);

	// update commands to drivers
	m_slaveArms[i].updateCmds(m_armCtrlCmds[i]);

END_FOR
END_METHOD

// state machine check and transit 
METHOD PROTECTED stateMachine : BOOL
VAR_IN_OUT CONSTANT
		i_slavesInputDataPool:ST_SlaveInputDataPool;
END_VAR
VAR
	i:INT;
END_VAR
FOR i:=1 TO g_sArmNum DO
	// State machine transit 
	CASE m_slaveArmState[i] OF
		// init
		SlaveArmState_Init:
			IF m_armCtrl[i].isFinished  THEN
				m_nextSlaveArmState[i]:=SlaveArmState_SelfCheck;
			END_IF

		//self check
		SlaveArmState_SelfCheck:
			IF m_armCtrl[i].isFinished  THEN
				m_nextSlaveArmState[i]:=SlaveArmState_Standby;
			END_IF
		
		//standby
		SlaveArmState_Standby:
			IF m_slaveArms[i].panelOn THEN
				m_nextSlaveArmState[i]:=SlaveArmState_MountPanel;
			END_IF
		
		//mount panel
		SlaveArmState_MountPanel:
			IF m_armCtrl[i]. isFinished THEN
				m_nextSlaveArmState[i]:=SlaveArmState_PanelReady;
				
				// NOTICE: multiple cycles joints back to center during initialization
				// 			need to reset joints encoder data again
				m_slaveArms[i].initJntPos();
			END_IF
		
		//panel ready
		SlaveArmState_PanelReady:
			IF m_slaveArms[i].instruOn THEN
				m_slaveArms[i].readInstruInfo();
				m_nextSlaveArmState[i]:=SlaveArmState_MountInstru;
			END_IF
			
(*		

		
		
		//mount instrument
		SlaveArmState_Mountnstru:
		
		//mount instrument
		SlaveArmState_Mountnstru:
		
		//instrument ready
		SlaveArmState_InstruReady:
		
		//master-slave control
		SlaveArmState_MasterSlave:
		
		//mount endoscope
		SlaveArmState_MountScope:
		
		//endoscope ready
		SlaveArmState_ScopeReady:
		
		//endoscope control
		SlaveArmState_EndoScope:
		
		//arm adjust
		SlaveArmState_Adjust:
		
		//cart control
		SlaveArmState_Cart:
*)
	END_CASE
	
	// Controller transit
	IF m_nextSlaveArmState[i]<> m_slaveArmState[i] THEN
		// reset current controller
		m_armCtrl[i].reset();
		
		// transit to new controller
		m_lastSlaveArmState[i]:=m_slaveArmState[i];
		m_slaveArmState[i]:=m_nextSlaveArmState[i];
		m_armCtrl[i]:=m_armCtrlFactory[i,m_slaveArmState[i]];
		
		// init next controller
		m_armCtrl[i].Init(m_slaveArms[i],m_armCtrlCmds[i]);
		m_slaveArms[i].updateCmds(m_armCtrlCmds[i]);
	END_IF
END_FOR
END_METHOD

END_FUNCTION_BLOCK

// ---- FBs_Robots/FB_SlaveArm.TcPOU
FUNCTION_BLOCK FB_SlaveArm
VAR_INPUT
END_VAR
VAR_OUTPUT
END_VAR
VAR
	// arm index, from 1 to 4
	m_armIdx: INT;
	
	// grip angle
	m_gripAngle :LREAL;
	
	// joints
	m_joints :ARRAY[1..g_sJntNum] OF FB_SlaveJoint;
	
	// panel and insturment  install signal
	m_panelInstrumentOnIO AT%I*	:UDINT;
	m_panelOnCounts :INT :=0;
	m_instruOnCounts :INT :=0;
	m_panelInstruOnCountThres :INT :=50;
	m_panelOnFlag :BOOL;
	m_instruOnFlag :BOOL;
	
	// adjust signal
	m_adjustIO AT%I* :UDINT;
	m_adjustOnCounts :INT :=0;
	m_adjustOnCountThres :INT :=50;
	m_adjustOnFlag :BOOL;
	
	// instrument instance
	m_instrument : FB_Instrument;

	// arm cartesian data, defined in each arm origin
	m_curCartPose	:ST_Frame;
	m_curCartTwist: Vec6d;
	
	// arm joint data
	m_curMotorPos :Vec8d;
	m_curLinkPos :Vec8d;
	m_curLinkSingle :Vec8d;
	m_curJntPos :Vec8d;
	m_curDHJntPos :Vec6d;
	m_curGripAngle :LREAL;
	m_curJntVel :Vec8d;
	m_curJntTrq :Vec8d;
	m_cmdJntTrq :Vec8d;
	m_rawJntCurrent :Vec8d;
	m_filtJntCurrent :Vec8d;
	m_cmdJntCurrent : Vec8d;
		
	// arm dynamic data
	m_jntGravity : Vec8d:=g_zeroVec8d;
	m_jntMassMat : Mat3d;
	
	// arm jacobian and inverse
	m_jaco : Mat6d;
	
	// simulated status
	m_simJntPos :Vec8d;
	m_simDHJntPos :Vec6d;
	m_simGripAngle :LREAL;
	m_simCartPose : ST_Frame;
	m_simJaco : Mat6d;
	m_simJacoInv :Mat6d;
	m_isSingularity:BOOL:=false;
	
	// joint position controller
	m_jntPIDCtrl :ARRAY[1..g_sJntNum] OF FB_PID;
	
	// code execute time measure
	m_codeTime : Profiler;
	
	m_ReadLDP:R_TRIG;
	ReadInfoIntrusStart:BOOL;
END_VAR

// check if adjust button is pressed
METHOD adjustDetect : BOOL
VAR_INPUT
END_VAR
// TODO: need to be reviewed
IF (m_adjustIO AND 16#0008)=8 THEN
	m_adjustOnCounts :=MIN(m_adjustOnCounts +1,m_adjustOnCountThres);
ELSE
	m_adjustOnCounts :=0;
END_IF

adjustDetect := m_adjustOnCounts >= m_adjustOnCountThres;
END_METHOD

PROPERTY adjustOn : bool
GET
adjustOn := m_adjustOnFlag;
END_GET
END_PROPERTY

PROPERTY armIdx : int
GET
armIdx:=m_armIdx;
END_GET
END_PROPERTY

METHOD PUBLIC calcJaco : BOOL
VAR_IN_OUT CONSTANT
	i_DHJntPos :Vec6d;
END_VAR
VAR_IN_OUT
	r_jaco :Mat6d;
END_VAR
VAR_INPUT
END_VAR

VAR
	d1, L, a, b :LREAL;
	q3:LREAL;

	c1,c2,c4,c5,c6,c7 :LREAL;
	s1,s2,s4,s5,s6,s7 :LREAL;
END_VAR
d1:=GVL_SlaveArmKinematic.g_d1;
L:=m_instrument.kinematicParameters.m_rodLength;
a:=m_instrument.kinematicParameters.m_headLength;
b:=m_instrument.kinematicParameters.m_fingerLenght;

q3:=i_DHJntPos[3];
q3:=i_DHJntPos[3];
c1:=COS(i_DHJntPos[1]);
c2:=COS(i_DHJntPos[2]);
c4:=COS(i_DHJntPos[4]);
c5:=COS(i_DHJntPos[5]);
c6:=COS(i_DHJntPos[6]);

s1:=SIN(i_DHJntPos[1]);
s2:=SIN(i_DHJntPos[2]);
s4:=SIN(i_DHJntPos[4]);
s5:=SIN(i_DHJntPos[5]);
s6:=SIN(i_DHJntPos[6]);

// jacobian with DH joints
r_jaco[1,1]:=b*(c6*(c5*(c1*s4 - c2*c4*s1) + s1*s2*s5) - s6*(c1*c4 + c2*s1*s4)) + a*(c5*(c1*s4 - c2*c4*s1) + s1*s2*s5) - L*s1*s2 + q3*s1*s2;
r_jaco[1,2]:=-c1*(a*(c2*s5 + c4*c5*s2) - L*c2 + q3*c2 + b*(c6*(c2*s5 + c4*c5*s2) + s2*s4*s6));
r_jaco[1,3]:=-c1*s2;
r_jaco[1,4]:=s1*s2*(a*(c2*s5 + c4*c5*s2) + b*(c6*(c2*s5 + c4*c5*s2) + s2*s4*s6)) - c2*(b*(c6*(c5*(c1*s4 - c2*c4*s1) + s1*s2*s5) - s6*(c1*c4 + c2*s1*s4)) + a*(c5*(c1*s4 - c2*c4*s1) + s1*s2*s5));
r_jaco[1,5]:=- (a*(c2*s5 + c4*c5*s2) + b*(c6*(c2*s5 + c4*c5*s2) + s2*s4*s6))*(c1*c4 + c2*s1*s4) - s2*s4*(b*(c6*(c5*(c1*s4 - c2*c4*s1) + s1*s2*s5) - s6*(c1*c4 + c2*s1*s4)) + a*(c5*(c1*s4 - c2*c4*s1) + s1*s2*s5));
r_jaco[1,6]:= b*(c6*(c5*(c1*s4 - c2*c4*s1) + s1*s2*s5) - s6*(c1*c4 + c2*s1*s4))*(c2*c5 - c4*s2*s5) + b*(s5*(c1*s4 - c2*c4*s1) - c5*s1*s2)*(c6*(c2*s5 + c4*c5*s2) + s2*s4*s6);


r_jaco[2,1]:=0;
r_jaco[2,2]:=c1*(a*(c5*(s1*s4 + c1*c2*c4) - c1*s2*s5) + b*(c6*(c5*(s1*s4 + c1*c2*c4) - c1*s2*s5) - s6*(c4*s1 - c1*c2*s4)) + L*c1*s2 - q3*c1*s2) - s1*(b*(c6*(c5*(c1*s4 - c2*c4*s1) + s1*s2*s5) - s6*(c1*c4 + c2*s1*s4)) + a*(c5*(c1*s4 - c2*c4*s1) + s1*s2*s5) - L*s1*s2 + q3*s1*s2);
r_jaco[2,3]:= c2;
r_jaco[2,4]:=- s1*s2*(a*(c5*(s1*s4 + c1*c2*c4) - c1*s2*s5) + b*(c6*(c5*(s1*s4 + c1*c2*c4) - c1*s2*s5) - s6*(c4*s1 - c1*c2*s4))) - c1*s2*(b*(c6*(c5*(c1*s4 - c2*c4*s1) + s1*s2*s5) - s6*(c1*c4 + c2*s1*s4)) + a*(c5*(c1*s4 - c2*c4*s1) + s1*s2*s5));
r_jaco[2,5]:=(a*(c5*(s1*s4 + c1*c2*c4) - c1*s2*s5) + b*(c6*(c5*(s1*s4 + c1*c2*c4) - c1*s2*s5) - s6*(c4*s1 - c1*c2*s4)))*(c1*c4 + c2*s1*s4) - (b*(c6*(c5*(c1*s4 - c2*c4*s1) + s1*s2*s5) - s6*(c1*c4 + c2*s1*s4)) + a*(c5*(c1*s4 - c2*c4*s1) + s1*s2*s5))*(c4*s1 - c1*c2*s4);
r_jaco[2,6]:=b*(c6*(c5*(c1*s4 - c2*c4*s1) + s1*s2*s5) - s6*(c1*c4 + c2*s1*s4))*(s5*(s1*s4 + c1*c2*c4) + c1*c5*s2) - b*(s5*(c1*s4 - c2*c4*s1) - c5*s1*s2)*(c6*(c5*(s1*s4 + c1*c2*c4) - c1*s2*s5) - s6*(c4*s1 - c1*c2*s4));

r_jaco[3,1]:=a*(c5*(s1*s4 + c1*c2*c4) - c1*s2*s5) + b*(c6*(c5*(s1*s4 + c1*c2*c4) - c1*s2*s5) - s6*(c4*s1 - c1*c2*s4)) + L*c1*s2 - q3*c1*s2;
r_jaco[3,2]:=-s1*(a*(c2*s5 + c4*c5*s2) - L*c2 + q3*c2 + b*(c6*(c2*s5 + c4*c5*s2) + s2*s4*s6));
r_jaco[3,3]:=-s1*s2;
r_jaco[3,4]:=- c2*(a*(c5*(s1*s4 + c1*c2*c4) - c1*s2*s5) + b*(c6*(c5*(s1*s4 + c1*c2*c4) - c1*s2*s5) - s6*(c4*s1 - c1*c2*s4))) - c1*s2*(a*(c2*s5 + c4*c5*s2) + b*(c6*(c2*s5 + c4*c5*s2) + s2*s4*s6));
r_jaco[3,5]:=- (a*(c2*s5 + c4*c5*s2) + b*(c6*(c2*s5 + c4*c5*s2) + s2*s4*s6))*(c4*s1 - c1*c2*s4) - s2*s4*(a*(c5*(s1*s4 + c1*c2*c4) - c1*s2*s5) + b*(c6*(c5*(s1*s4 + c1*c2*c4) - c1*s2*s5) - s6*(c4*s1 - c1*c2*s4)));
r_jaco[3,6]:=b*(c6*(c5*(s1*s4 + c1*c2*c4) - c1*s2*s5) - s6*(c4*s1 - c1*c2*s4))*(c2*c5 - c4*s2*s5) + b*(c6*(c2*s5 + c4*c5*s2) + s2*s4*s6)*(s5*(s1*s4 + c1*c2*c4) + c1*c5*s2);

r_jaco[4,1]:=0;
r_jaco[4,2]:=-s1;
r_jaco[4,3]:=0;
r_jaco[4,4]:=-c1*s2;
r_jaco[4,5]:=c1*c2*s4 - c4*s1;
r_jaco[4,6]:=s5*(s1*s4 + c1*c2*c4) + c1*c5*s2;

r_jaco[5,1]:=-1;
r_jaco[5,2]:=0;
r_jaco[5,3]:=0;
r_jaco[5,4]:=c2;
r_jaco[5,5]:=s2*s4;
r_jaco[5,6]:=c4*s2*s5 - c2*c5;

r_jaco[6,1]:=0;
r_jaco[6,2]:=c1;
r_jaco[6,3]:=0;
r_jaco[6,4]:=-s1*s2;
r_jaco[6,5]:=c1*c4 + c2*s1*s4;
r_jaco[6,6]:=c5*s1*s2 - s5*(c1*s4 - c2*c4*s1);
END_METHOD

METHOD checkIO : BOOL
VAR_INPUT
END_VAR
// check adjust button
m_adjustOnFlag := adjustDetect();
// check panel and instrument
m_panelOnFlag := panelDetect();
m_instruOnFlag := instruDetect();
IF FALSE = m_instruOnFlag THEN
	ReadInfoIntrusStart:=FALSE;
	m_instrument.reset();
ELSIF InstruType_UNKNOWM = m_instrument.InstruReadPara.m_Instrutype THEN
	ReadInfoIntrusStart:=TRUE;
	m_instrument.readParameters();
END_IF

m_ReadLDP(CLK:= ReadInfoIntrusStart, Q=>m_instrument.InstruReadPara.i_ReadInfoIntrus );
//m_instruOnFlag := m_instruOnFlag AND (m_instrument.InstruReadPara.m_Instrutype <> InstruType_UNKNOWM);
END_METHOD

PROPERTY cmdJntCurrent : REFERENCE TO  Vec8d
GET
cmdJntCurrent ref= m_cmdJntCurrent;
END_GET
END_PROPERTY

PROPERTY curCartPose : REFERENCE TO ST_Frame
GET
curCartPose ref=m_curCartPose;
END_GET
END_PROPERTY

PROPERTY curCartTwist : REFERENCE TO Vec6d
GET
curCartTwist ref=m_curCartTwist;
END_GET
END_PROPERTY

PROPERTY curJntPos : REFERENCE TO Vec8d
GET
curJntPos ref=m_curJntPos;
END_GET
END_PROPERTY

PROPERTY curJntTrq : REFERENCE TO Vec8d
GET
curJntTrq ref=m_curJntTrq;
END_GET
END_PROPERTY

PROPERTY curJntVel :REFERENCE TO Vec8d
GET
curJntVel ref=m_curJntVel;
END_GET
END_PROPERTY

PROPERTY curLinkPos :REFERENCE TO Vec8d
GET
curLinkPos ref=m_curLinkPos;
END_GET
END_PROPERTY

PROPERTY curMotorPos : REFERENCE TO  Vec8d
GET
curMotorPos ref=m_curMotorPos;
END_GET
END_PROPERTY

METHOD PUBLIC enable : BOOL
VAR_IN_OUT CONSTANT
	i_jntIdx :Vec8i;
END_VAR
VAR
	i :INT ;
END_VAR
FOR i:=1 TO g_sJntNum DO
	IF 1= i_jntIdx[i] THEN
		m_joints[i].enable();
	ELSE
		m_joints[i].disable();
	END_IF
END_FOR
END_METHOD

PROPERTY filtJntCurrent :REFERENCE TO Vec8d
GET
filtJntCurrent ref= m_filtJntCurrent;
END_GET
END_PROPERTY

// from active joint position to cartesian pose in arm origin
METHOD PROTECTED forwardKinematic : BOOL
VAR_IN_OUT CONSTANT
	i_DHJntPos :Vec6d;
END_VAR
VAR_IN_OUT
	r_cartPose :ST_Frame;
	r_gripAngle : LREAL;
END_VAR
VAR
	d1, L, a, b :LREAL;
	q3 :LREAL;

	c1,c2,c4,c5,c6,c7 :LREAL;
	s1,s2,s4,s5,s6,s7 :LREAL;

END_VAR

d1:=GVL_SlaveArmKinematic.g_d1;
L:=m_instrument.kinematicParameters.m_rodLength;
a:=m_instrument.kinematicParameters.m_headLength;
b:=m_instrument.kinematicParameters.m_fingerLenght;

q3:=i_DHJntPos[3];
c1:=COS(i_DHJntPos[1]);
c2:=COS(i_DHJntPos[2]);
c4:=COS(i_DHJntPos[4]);
c5:=COS(i_DHJntPos[5]);
c6:=COS(i_DHJntPos[6]);

s1:=SIN(i_DHJntPos[1]);
s2:=SIN(i_DHJntPos[2]);
s4:=SIN(i_DHJntPos[4]);
s5:=SIN(i_DHJntPos[5]);
s6:=SIN(i_DHJntPos[6]);


// cartesian pose frame
r_cartPose.m_pos[1]:=a*(c5*(s1*s4 + c1*c2*c4) - c1*s2*s5) + b*(c6*(c5*(s1*s4 + c1*c2*c4) - c1*s2*s5) - s6*(c4*s1 - c1*c2*s4)) + L*c1*s2 - q3*c1*s2;
r_cartPose.m_pos[2]:=a*(c2*s5 + c4*c5*s2) - d1 - L*c2 + q3*c2 + b*(c6*(c2*s5 + c4*c5*s2) + s2*s4*s6);
r_cartPose.m_pos[3]:=L*s1*s2 - a*(c5*(c1*s4 - c2*c4*s1) + s1*s2*s5) - b*(c6*(c5*(c1*s4 - c2*c4*s1) + s1*s2*s5) - s6*(c1*c4 + c2*s1*s4)) - q3*s1*s2;

r_cartPose.m_rot[1,1]:= c6*(c5*(s1*s4 + c1*c2*c4) - c1*s2*s5) - s6*(c4*s1 - c1*c2*s4);
r_cartPose.m_rot[2,1]:=c6*(c2*s5 + c4*c5*s2) + s2*s4*s6;
r_cartPose.m_rot[3,1]:=s6*(c1*c4 + c2*s1*s4) - c6*(c5*(c1*s4 - c2*c4*s1) + s1*s2*s5);

r_cartPose.m_rot[1,2]:=- s6*(c5*(s1*s4 + c1*c2*c4) - c1*s2*s5) - c6*(c4*s1 - c1*c2*s4);
r_cartPose.m_rot[2,2]:=c6*s2*s4 - s6*(c2*s5 + c4*c5*s2);
r_cartPose.m_rot[3,2]:=s6*(c5*(c1*s4 - c2*c4*s1) + s1*s2*s5) + c6*(c1*c4 + c2*s1*s4);

r_cartPose.m_rot[1,3]:= s5*(s1*s4 + c1*c2*c4) + c1*c5*s2;
r_cartPose.m_rot[2,3]:= c4*s2*s5 - c2*c5;
r_cartPose.m_rot[3,3]:=c5*s1*s2 - s5*(c1*s4 - c2*c4*s1);
END_METHOD

PROPERTY gripAngle : LREAL
GET
gripAngle:=m_gripAngle;
END_GET
END_PROPERTY

METHOD PUBLIC init : BOOL
VAR_INPUT
	i_armIdx:INT;
END_VAR
VAR 
	i :INT ;
	currentRatioMotor2Jnt: LREAL;
END_VAR
// arm statues init
m_armIdx:=i_armIdx;
m_gripAngle:=0;

// joint init
FOR i:=1 TO g_sJntNum DO
	IF i<4 THEN
		m_joints[i].init(m_armIdx, i,g_slaveArmCtrlCycleTime, 1);
	ELSE
		m_joints[i].init(m_armIdx, i,g_slaveArmCtrlCycleTime, 4);
	END_IF
END_FOR

// init joint encoder and position calculation
initJntPos();

// joint controller init
FOR i:=1 TO g_sJntNum DO 
	currentRatioMotor2Jnt:=GVL_SlaveMotorParameters.g_motorTrqConst[i]*GVL_SlaveMotorParameters.g_motorReduction[i]/1000;
	m_jntPIDCtrl[i].init(g_slaveArmCtrlCycleTime,GVL_slaveControlParameters.g_posKp[i],GVL_slaveControlParameters.g_posKd[i],
		GVL_slaveControlParameters.g_posKi[i], GVL_slaveControlParameters.g_posKiLimit[i]* currentRatioMotor2Jnt,
		GVL_slaveControlParameters.g_posCtrlLimit[i]*currentRatioMotor2Jnt);
END_FOR
END_METHOD

METHOD initJntPos : BOOL
VAR_INPUT
END_VAR
VAR
	i:INT ;
END_VAR
// joint init
FOR i:=1 TO g_sJntNum DO
	m_joints[i].initJntPos();
END_FOR


// update arm status if joint position is re-init
updateStatus();
END_METHOD

// check if instrument is on
METHOD instruDetect : BOOL
VAR_INPUT
END_VAR
// TODO: need to be reviewed
//Instrument single   At installation--2#0*0*   not installation --2#1*1*  And Hall single --2#100 0000
IF (m_panelInstrumentOnIO AND 16#4A) = 64  THEN
	m_instruOnCounts := MIN( m_instruOnCounts +1,m_panelInstruOnCountThres);
ELSIF (m_panelInstrumentOnIO AND 16#4A) = 10  THEN
	m_instruOnCounts :=0;
END_IF

instruDetect := m_instruOnCounts >= m_panelInstruOnCountThres;
END_METHOD

PROPERTY instrument : REFERENCE TO FB_Instrument
GET
instrument REF=m_instrument;
END_GET
END_PROPERTY

PROPERTY instruOn : bool
GET
instruOn:=m_instruOnFlag;
END_GET
END_PROPERTY

METHOD PUBLIC isEnabled : BOOL
VAR_IN_OUT CONSTANT
	i_jntIdx :Vec8i;
END_VAR
VAR
	i :INT ;
END_VAR
isEnabled := TRUE;
FOR i:=1 TO g_sJntNum DO
	IF 1= i_jntIdx[i] THEN
		isEnabled :=  (m_joints[i].isEnabled() AND isEnabled);
	END_IF
END_FOR
END_METHOD

PROPERTY isSingurality : bool
GET
isSingurality:=m_isSingularity;
END_GET
END_PROPERTY

PROPERTY jaco :REFERENCE TO Mat6d
GET
jaco ref= m_jaco;
END_GET
END_PROPERTY

PROPERTY jntGravity :REFERENCE TO Vec8d
GET
jntGravity ref=m_jntGravity;
END_GET
END_PROPERTY

PROPERTY linkSingle :REFERENCE TO Vec8d
GET
linkSingle ref=m_curLinkSingle;
END_GET
END_PROPERTY

PROPERTY PUBLIC massMat :REFERENCE TO Mat3d
GET
massMat ref=m_jntMassMat;
END_GET
END_PROPERTY

// check if panel is on
METHOD panelDetect : BOOL
VAR_INPUT
END_VAR
// TODO: need to be reviewed
//Panel single  At installation--2#0000   not installation --2#0101
IF (m_panelInstrumentOnIO AND 16#05) = 0 THEN
	m_panelOnCounts := MIN( m_panelOnCounts +1,m_panelInstruOnCountThres);
ELSIF (m_panelInstrumentOnIO AND 16#05) = 5  THEN
	m_panelOnCounts :=0;
END_IF

panelDetect := m_panelOnCounts >= m_panelInstruOnCountThres;
END_METHOD

PROPERTY panelOn : bool
GET
panelOn :=m_panelOnFlag;
END_GET
END_PROPERTY

PROPERTY rawJntCurrent :REFERENCE TO Vec8d
GET
rawJntCurrent ref=m_rawJntCurrent;
END_GET
END_PROPERTY

METHOD readInstruInfo : BOOL
VAR_INPUT
END_VAR
m_instrument.readParameters();
END_METHOD

PROPERTY simCartPose :REFERENCE TO ST_Frame
GET
simCartPose:=m_simCartPose;
END_GET
END_PROPERTY

PROPERTY simJaco :REFERENCE TO mat6d
GET
simJaco:=m_simJaco;
END_GET
END_PROPERTY

// update joints control command
METHOD PUBLIC updateCmds : BOOL
VAR_IN_OUT CONSTANT
	i_armCtrlCmd : ST_SlaveArmCtrlCmds;
END_VAR
VAR
	i:INT;
END_VAR
m_cmdJntTrq:=i_armCtrlCmd.m_cmdJntTrq;
m_simJntPos:=i_armCtrlCmd.m_cmdJntPos;

// update simulated master arm
updateSimStatus();

// enable/disable joints
enable(i_armCtrlCmd.m_jntEnableFlag);

	m_codeTime(START:=TRUE, RESET:=TRUE);
// position/torque control
FOR i:=1 TO g_sJntNum DO 
	IF i_armCtrlCmd.m_jntOPMode[i]=DriverOPMode_PosTrq THEN
		// position controller and gravity feedforward
		m_cmdJntTrq[i]:=m_jntPIDCtrl[i].run(i_armCtrlCmd.m_cmdJntPos[i],m_curJntPos[i],i_armCtrlCmd.m_cmdJntVel[i],m_curJntVel[i]);
		m_cmdJntTrq[i]:=m_cmdJntTrq[i]+m_jntGravity[i];
		m_joints[i].updateCmds(DriverOPMode_Trq,i_armCtrlCmd.m_cmdJntPos[i],m_cmdJntTrq[i]);
	ELSIF i_armCtrlCmd.m_jntOPMode[i]=DriverOPMode_Trq THEN
		// gravity feedforward
		m_cmdJntTrq[i]:=m_cmdJntTrq[i]+m_jntGravity[i];
		m_joints[i].updateCmds(DriverOPMode_Trq,i_armCtrlCmd.m_cmdJntPos[i],m_cmdJntTrq[i]);
	ELSE
		m_jntPIDCtrl[i].reset();
		m_cmdJntTrq[i]:=0;
		m_joints[i].updateCmds(DriverOPMode_Pos,i_armCtrlCmd.m_cmdJntPos[i],m_cmdJntTrq[i]);
	END_IF
	
END_FOR
	m_codeTime(START:=False);
END_METHOD

METHOD PUBLIC updateDyna : BOOL
VAR_IN_out constant
	slaveDynaData : ST_SlaveDynaData;
END_VAR
m_jntMassMat:=slaveDynaData.m_massMat[m_armIdx];
m_jntGravity[1]:=slaveDynaData.m_gravity[m_armIdx][1];
m_jntGravity[2]:=slaveDynaData.m_gravity[m_armIdx][2];
m_jntGravity[3]:=slaveDynaData.m_gravity[m_armIdx][3];
END_METHOD

METHOD PUBLIC updateSimStatus : BOOL
VAR_INPUT
END_VAR
//IF m_instrument.ready THEN
	// instrument kinematic
	m_instrument.instruFK(m_simJntPos, m_simDHJntPos, m_simGripAngle);

	// simulated cartesion pose 
	forwardKinematic(m_simDHJntPos,m_simCartPose,m_simGripAngle);
	
	// simulated jacobian
	calcJaco(m_simDHJntPos,m_simJaco);
	m_isSingularity:=NOT(invMat6(m_simJaco, m_simJacoInv));
//END_IF
END_METHOD

// update arm status, including kinematic and dynamic
METHOD PUBLIC updateStatus : BOOL
VAR_INPUT
END_VAR
VAR 
	i,j:INT;
END_VAR
// update joint data
FOR i:=1 TO g_sJntNum DO
	m_joints[i].updateStatus();
END_FOR

// check panel and instrument
checkIO();

// get joint data
FOR i:=1 TO g_sJntNum DO
	m_curMotorPos[i]:=m_joints[i].motorPos;
	m_curLinkPos[i]:=m_joints[i].linkPos;
	m_curLinkSingle[i]:=m_joints[i].linkSingle;
	m_curJntPos[i]:=m_joints[i].jntPos;
	m_curJntVel[i]:=m_joints[i].jntVel;
	m_curJntTrq[i]:=m_joints[i].jntTrq;
	m_rawJntCurrent[i]:=m_joints[i].rawCurrent;
	m_filtJntCurrent[i]:=m_joints[i].filtCurrent;
	m_cmdJntCurrent[i]:=m_joints[i].cmdCurrent;
END_FOR 

// only update carteisn data when instrument is ready
//IF m_instrument.ready THEN
	
	// instrument kinematic
	m_instrument.instruFK(m_curJntPos, m_curDHJntPos, m_curGripAngle);

	// cartesion pose
	forwardKinematic(m_curDHJntPos,m_curCartPose,m_gripAngle);
	
	// jacobian
	calcJaco(m_curDHJntPos,m_jaco);
	
	// cartesian twist
//END_IF
END_METHOD

END_FUNCTION_BLOCK

// ---- FBs_Robots/FB_SlaveJoint.TcPOU
FUNCTION_BLOCK FB_SlaveJoint EXTENDS FB_JointBase
VAR_INPUT
END_VAR
VAR_OUTPUT
END_VAR
VAR
END_VAR

METHOD init : BOOL
VAR_INPUT
	i_armIdx :INT;
	i_jntIdx :INT;
	i_controlCycleTime :LREAL;
	// velocity is calculated every (m_velCalcCycles) control cycles
	// TODO: insturment joint motor can not reach 4k now, so calculate their velocity with 1k frequency, need to remove later
	i_velCalcCycles :INT;
END_VAR
m_armIdx:=i_armIdx;
m_jntIdx:=i_jntIdx;
m_cycleTime := i_controlCycleTime;
m_velCalcCycles :=MAX(i_velCalcCycles,1);

// hardware parameters
m_motorEncoderRes :=GVL_SlaveMotorParameters.g_incEncoderRes[i_jntIdx];
m_linkEncoderRes :=GVL_SlaveMotorParameters.g_absEncoderRes[i_jntIdx];
m_motorReduction :=GVL_SlaveMotorParameters.g_motorReduction[i_jntIdx];
m_linkEncoderReduction :=GVL_SlaveMotorParameters.g_absEncoderReduction[i_jntIdx];
m_trqConst :=GVL_SlaveMotorParameters.g_motorTrqConst[i_jntIdx];
m_maxCurrent :=GVL_SlaveMotorParameters.g_motorMaxCurrent[i_jntIdx];
m_motorDir :=GVL_SlaveMotorParameters.g_motorDir[i_jntIdx];								
m_minJntPos	:=GVL_SlaveMotorParameters.g_minJntPos[i_jntIdx];
m_maxJntPos	:=GVL_SlaveMotorParameters.g_maxJntPos[i_jntIdx];

//link encoder calibartion data
m_linkEncoderDir :=GVL_SlaveJointEncoderCaliData.g_asbEncoderDir[i_jntIdx];
m_minLinkEncoder :=GVL_SlaveJointEncoderCaliData.g_minLinkEncoder[i_armIdx, i_jntIdx] - m_linkEncoderDir*GVL_SlaveJointEncoderCaliData.g_linkEncLimitBuffer; // expand limit
m_maxLinkEncoder :=GVL_SlaveJointEncoderCaliData.g_maxLinkEncoder[i_armIdx, i_jntIdx] + m_linkEncoderDir*GVL_SlaveJointEncoderCaliData.g_linkEncLimitBuffer; // expand limit
m_caliLinkEncoder :=GVL_SlaveJointEncoderCaliData.g_caliLinkEncoder[i_armIdx, i_jntIdx];
m_linkEncCaliJntPos :=GVL_SlaveJointEncoderCaliData.g_linkEncCaliJntPos[i_jntIdx];
m_linkEncZeroCross :=GVL_SlaveJointEncoderCaliData.g_linkEncZeroCross[i_armIdx, i_jntIdx];
m_multiCycles :=GVL_SlaveJointEncoderCaliData.g_multipleCyclesJoint[i_armIdx,i_jntIdx];

// convert cali link encoder if joint cross zero
IF 1=m_linkEncZeroCross THEN
	IF 1=m_linkEncoderDir AND m_caliLinkEncoder < m_minLinkEncoder THEN
		m_caliLinkEncoder := GVL_SlaveJointEncoderCaliData.g_caliLinkEncoder[i_armIdx, i_jntIdx] + m_linkEncoderRes;
	ELSIF -1=m_linkEncoderDir AND m_caliLinkEncoder < m_maxLinkEncoder THEN
		m_caliLinkEncoder := GVL_SlaveJointEncoderCaliData.g_caliLinkEncoder[i_armIdx, i_jntIdx] + m_linkEncoderRes;
	END_IF
END_IF

// macro data
m_trq2CurrentRatio:=m_motorDir * 1000.0/(m_trqConst*m_motorReduction);
m_current2TrqRatio:=m_motorDir * (m_trqConst*m_motorReduction)/1000.0;
m_linkEnc2PosRatio := 2*PI*m_linkEncoderDir/(m_linkEncoderReduction*m_linkEncoderRes);
m_motorEnc2PosRatio := 2*PI * m_motorDir/(m_motorReduction * m_motorEncoderRes);

// motor data init
m_curJntVel:=0;
m_curJntTrq :=0;
m_rawCurrent :=0;
m_filtCurrent :=0;
m_cmdJntVel :=0.0;
m_cmdJntTrq :=0.0;
m_cmdCurrent := 0.0;

// filter init
m_jntVelLpf.init(1, GVL_SlaveControlParameters.g_curJntVelLpfCutoffFreq, g_slaveArmCtrlFreq/m_velCalcCycles);
m_cmdTrqLpf.init(1, GVL_SlaveControlParameters.g_cmdJntTrqLpfCutoffFreq, g_slaveArmCtrlFreq);
m_curTrqLpf.init(1, GVL_SlaveControlParameters.g_curJntTrqLpfCutoffFreq, g_slaveArmCtrlFreq);

// driver init value
m_motorOutputs.m_controlWord:=DriverCtrlWord_INIT;
m_motorOutputs.m_opMode:=INT_TO_SINT(DriverOPMode_Pos);
m_motorOutputs.m_cmdCurrent:=0;
m_motorOutputs.m_cmdMotorEncoder:=m_motorInputs.m_motorEncoder;
m_motorOutputs.m_ratedCurrent:=200;
END_METHOD

METHOD PUBLIC updateCmds : BOOL
VAR_INPUT
	i_opMode : E_DriverOPMode;
	i_cmdPos :LREAL;
	i_cmdTrq :LREAL;
END_VAR
VAR
	filtCmdTrq :LREAL;
END_VAR
SUPER^.updateCmds(i_opMode, i_cmdPos, i_cmdTrq);

// write SDO data
writeSDOData();
END_METHOD

METHOD PROTECTED writeSDOData : BOOL
VAR_INPUT
END_VAR
VAR
	SDOSubIndexMode :WORD;
	SDOSubIndexCur :WORD;
END_VAR
//动力盒移动关节和器械旋转关节，共享一个控制字，由SDO写入
IF (m_jntIdx=3) OR (m_jntIdx=8)  THEN
	SDOSubIndexMode :=16#609B;
	SDOSubIndexCur:=16#6098;
//动力盒3、5号电机为一个驱动器，共享一个控制字，由SDO写入
ELSIF (m_jntIdx=4) OR (m_jntIdx=6)  THEN
	SDOSubIndexMode :=16#609C;
	SDOSubIndexCur:=16#6099;
//动力盒2、4号电机为一个驱动器，共享一个控制字，由SDO写入
ELSIF (m_jntIdx=5) OR (m_jntIdx=7)  THEN
	SDOSubIndexMode :=16#609D;
	SDOSubIndexCur:=16#609A;
END_IF

IF m_jntIdx <3 THEN
	RETURN;
END_IF

m_opModeSDOWrite(sNetID:= GVL_SlaveMotorParameters.g_slaveArmNetID[m_armIdx],
				nSlaveAddr := GVL_SlaveMotorParameters.g_slaveJointNetPort[m_armIdx,m_jntIdx],
				nSubIndex:=0,nIndex:=SDOSubIndexMode,pSrcBuf:=ADR(m_motorOutputs.m_opMode),cbBufLen:=SIZEOF(m_motorOutputs.m_opMode),bExecute:=TRUE);
IF NOT m_opModeSDOWrite.bBusy THEN
	m_opModeSDOWrite(bExecute:=FALSE);
END_IF
	
m_MotorCurrentSDOWrite(sNetID:= GVL_SlaveMotorParameters.g_slaveArmNetID[m_armIdx],
				nSlaveAddr := GVL_SlaveMotorParameters.g_slaveJointNetPort[m_armIdx,m_jntIdx],
				nSubIndex:=0,nIndex:=SDOSubIndexCur,pSrcBuf:=ADR(m_motorOutputs.m_ratedCurrent),cbBufLen:=SIZEOF(m_motorOutputs.m_ratedCurrent),bExecute:=TRUE);
IF NOT m_opModeSDOWrite.bBusy THEN
	m_opModeSDOWrite(bExecute:=FALSE);
END_IF
END_METHOD

END_FUNCTION_BLOCK

// ---- FBs_Robots/FB_JointBase.TcPOU
FUNCTION_BLOCK FB_JointBase
VAR_INPUT
END_VAR
VAR_OUTPUT
END_VAR
VAR
	// arm and joint index
	m_armIdx :INT;
	m_jntIdx :INT;
	
	// motor IO
	m_motorInputs AT%I*	:ST_MotorInputs;
	m_motorOutputs AT%Q* :ST_MotorOutputs;
	
	// cycle time
	m_cycleTime :LREAL;
	
	// calibrated link encoder data
	m_minLinkEncoder :DINT;
	m_maxLinkEncoder :DINT;
	m_caliLinkEncoder :DINT;
	m_linkEncCaliJntPos :LREAL;
	m_linkEncZeroCross :INT;
	m_initMotorEnc : DINT;
	m_multiCycles :INT;
	
	// joint position from link encoder after power on
	m_initLinkPos :LREAL;
	
	// data for link encoder multiple cycles
	m_lastLinkEncoder :DINT;
	m_linkEncCycles:INT;
	
	// device paramters
	m_motorEncoderRes :DINT;
	m_linkEncoderRes :DINT;
	m_motorReduction :LREAL;
	m_linkEncoderReduction :LREAL;
	m_trqConst :LREAL;
	m_maxCurrent :LREAL;
	m_motorDir :INT;								
	m_linkEncoderDir :INT;
	m_minJntPos: LREAL;
	m_maxJntPos: LREAL;
	
	// macro defined data for quick calculation
	m_trq2CurrentRatio:LREAL;
	m_current2TrqRatio:LREAL;
	m_linkEnc2PosRatio :LREAL;
	m_motorEnc2PosRatio :LREAL;
	
	// joint data
	m_curMotorPos :LREAL;
	m_curLinkPos :LREAL;
	m_curJntPos	:LREAL;
	m_curJntVel :LREAL;
	m_curJntTrq :	LREAL;
	m_rawCurrent : LREAL;
	m_filtCurrent : LREAL;
	m_cmdJntPos :LREAL;
	m_cmdJntVel :LREAL;
	m_cmdJntTrq :LREAL;
	m_cmdCurrent : LREAL;
	m_lastJntPos :LREAL;
	
	// velocity filter
	m_jntVelLpf :FB_LowPassFilter;
	
	// command torque filter
	m_curTrqLpf : FB_LowPassFilter;
	m_cmdTrqLpf :FB_LowPassFilter;
	
	// velocity is calculated every (m_velCalcCycles) control cycles
	// TODO: insturment joint motor can not reach 4k now, so calculate their velocity with 1k frequency, need to remove later
	m_velCalcCycles :INT :=1;
	m_curVelCalCycles :INT :=1;
	
	// SDO writer
	m_opModeSDOWrite:FB_EcCoESdoWrite;
END_VAR

PROPERTY cmdCurrent : LREAL
GET
cmdCurrent:=m_cmdCurrent;
END_GET
END_PROPERTY

METHOD PUBLIC disable : BOOL
VAR_INPUT
END_VAR
m_motorOutputs.m_controlWord:=DriverCtrlWord_INIT;
disable:=true;
END_METHOD

METHOD PUBLIC enable : BOOL
VAR_INPUT
END_VAR
IF DriverStatusWord_INIT = m_motorInputs.m_statusWord THEN
	m_motorOutputs.m_controlWord:=DriverCtrlWord_PREOP;
	enable := FALSE;
ELSIF DriverStatusWord_PREOP = m_motorInputs.m_statusWord THEN
	m_motorOutputs.m_controlWord:=DriverCtrlWord_OP;
	enable :=  FALSE;
ELSIF DriverStatusWord_OP = m_motorInputs.m_statusWord THEN
	enable :=  TRUE;
//ELSE
//	m_motorOutputs.m_controlWord:=DriverCtrlWord_INIT;
//	enable :=  FALSE;
END_IF
END_METHOD

PROPERTY filtCurrent : LREAL
GET
filtCurrent:=m_filtCurrent;
END_GET
END_PROPERTY

METHOD initJntPos : BOOL
VAR_INPUT
END_VAR
m_lastLinkEncoder :=m_motorInputs.m_linkEncoder;
m_linkEncCycles:=0;
m_curLinkPos :=linkEnc2Pos();
m_initLinkPos:=m_curLinkPos;
m_initMotorEnc :=m_motorInputs.m_motorEncoder;
m_curMotorPos:=motorEnc2Pos();
m_curJntPos := m_curMotorPos;
m_cmdJntPos :=m_curJntPos;	
m_lastJntPos :=m_curJntPos;
END_METHOD

PROPERTY initLinkPos : lreal
GET
initLinkPos:=m_initLinkPos;
END_GET
SET
m_initLinkPos:=initLinkPos;
END_SET
END_PROPERTY

METHOD isEnabled : BOOL
VAR_INPUT
END_VAR
isEnabled :=(DriverStatusWord_OP = m_motorInputs.m_statusWord);
END_METHOD

PROPERTY jntPos : LREAL
GET
jntPos := m_curJntPos;
END_GET
END_PROPERTY

PROPERTY jntTrq : LREAL
GET
jntTrq:=m_curJntTrq;
END_GET
END_PROPERTY

PROPERTY jntVel : LREAL
GET
jntVel := m_curJntVel;
END_GET
END_PROPERTY

METHOD PROTECTED linkEnc2Pos : LREAL
VAR_INPUT
END_VAR
VAR
	incLinkPos :LREAL;
	newLinkEnc :DINT;
END_VAR
// cycle check
IF 1=m_multiCycles THEN
	IF (m_motorInputs.m_linkEncoder - m_lastLinkEncoder)*m_linkEncoderDir < -m_linkEncoderRes/2 THEN
		m_linkEncCycles :=m_linkEncCycles+1;
	ELSIF (m_motorInputs.m_linkEncoder - m_lastLinkEncoder)*m_linkEncoderDir > m_linkEncoderRes/2 THEN
		m_linkEncCycles :=m_linkEncCycles-1;
	END_IF
END_IF
m_lastLinkEncoder:=m_motorInputs.m_linkEncoder;

// convert link encoder if joint cross zero
newLinkEnc := m_motorInputs.m_linkEncoder;
IF 1=m_linkEncZeroCross AND 0 = m_multiCycles THEN
	IF 1=m_linkEncoderDir AND m_motorInputs.m_linkEncoder < m_minLinkEncoder THEN
		newLinkEnc := m_motorInputs.m_linkEncoder + m_linkEncoderRes;
	ELSIF -1=m_linkEncoderDir AND m_motorInputs.m_linkEncoder < m_maxLinkEncoder THEN
		newLinkEnc := m_motorInputs.m_linkEncoder + m_linkEncoderRes;
	END_IF
END_IF

// motion from calibrated points
incLinkPos := (newLinkEnc-m_caliLinkEncoder)*m_linkEnc2PosRatio;

// absolute joint position
linkEnc2Pos := incLinkPos + m_linkEncCaliJntPos + 2*PI* m_linkEncCycles;
END_METHOD

PROPERTY PUBLIC linkPos : LREAL
GET
linkPos:=m_curLinkPos;
END_GET
END_PROPERTY

METHOD PUBLIC motorEnc2Pos : LREAL
VAR_INPUT
END_VAR
motorEnc2Pos:= (m_motorInputs.m_motorEncoder-m_initMotorEnc)* m_motorEnc2PosRatio +m_initLinkPos;
END_METHOD

PROPERTY PUBLIC motorPos : LREAL
GET
motorPos := m_curMotorPos;
END_GET
END_PROPERTY

METHOD PROTECTED motorPos2Enc : DINT
VAR_INPUT
	i_jntPos :LREAL;
END_VAR

VAR
END_VAR
motorPos2Enc := LREAL_TO_DINT((i_jntPos-m_initLinkPos)/m_motorEnc2PosRatio + m_initMotorEnc);
END_METHOD

PROPERTY rawCurrent : LREAL
GET
rawCurrent := m_rawCurrent;
END_GET
END_PROPERTY

METHOD PUBLIC updateCmds : BOOL
VAR_INPUT
	i_opMode : E_DriverOPMode;
	i_cmdPos :LREAL;
	i_cmdTrq :LREAL;
END_VAR
VAR
	filtCmdTrq :LREAL;
END_VAR
m_motorOutputs.m_opMode:=INT_TO_SINT( i_opMode);
// pos mode
IF i_opMode = DriverOPMode_Pos THEN
	m_motorOutputs.m_cmdCurrent:=0;
	m_cmdTrqLpf.reset();	
//	i_cmdPos:=LIMIT(m_minJntPos, i_cmdPos, m_maxJntPos);
	m_motorOutputs.m_cmdMotorEncoder :=motorPos2Enc(i_cmdPos);
ELSIF i_opMode = DriverOPMode_Trq THEN
	filtCmdTrq:=m_cmdTrqLpf.run(i_cmdTrq);
	m_motorOutputs.m_cmdCurrent:=LREAL_TO_DINT(LIMIT(-m_maxCurrent, filtCmdTrq*m_trq2CurrentRatio,m_maxCurrent));
	m_motorOutputs.m_cmdMotorEncoder :=m_motorInputs.m_motorEncoder; 
END_IF
m_cmdCurrent:=m_motorOutputs.m_cmdCurrent;
END_METHOD

METHOD PUBLIC updateStatus : BOOL
VAR_INPUT
END_VAR
// compute joint position
m_curLinkPos:= linkEnc2Pos();
m_curMotorPos:=motorEnc2Pos();
m_curJntPos := m_curMotorPos;

// compute joint velocity
m_curVelCalCycles := m_curVelCalCycles+1;
IF m_curVelCalCycles > m_velCalcCycles THEN
	m_curJntVel:= (m_curJntPos-m_lastJntPos)/(m_cycleTime*m_velCalcCycles);
	m_curJntVel := m_jntVelLpf.run(m_curJntVel);
	m_lastJntPos :=m_curJntPos;	
	m_curVelCalCycles:=1;
END_IF


// current and torque
m_rawCurrent := m_motorInputs.m_current;
m_filtCurrent := m_curTrqLpf.run(m_rawCurrent);
m_curJntTrq := m_filtCurrent * m_current2TrqRatio;
END_METHOD

END_FUNCTION_BLOCK

// ---- FBs_Robots/FB_Instrument.TcPOU
FUNCTION_BLOCK FB_Instrument
VAR_INPUT
END_VAR
VAR_OUTPUT
END_VAR
VAR
	// ID
	m_ID: INT:=0;
	
	// series number
	m_seriesNum : ULINT:=0;
	
	// instrument type
	m_type : E_InstrumentType := InstruType_UNKNOWM;
	
	// current and max usage counts
	m_usageCounts :INT;
	m_maxUsageCounts :INT;
	
	// kinematic parameters	
	m_kinematicParameters:ST_InstruParameters; 
	
END_VAR

METHOD gripperAngleForwardTransform_ID12 : BOOL
VAR_INPUT
	frontAngle:LREAL;
END_VAR
VAR_OUTPUT
	endAngle:LREAL;
	Succeed:BOOL;
END_VAR
VAR
	minFrontAng :LREAL  := 16.6*2*g_deg2Rad;
	maxFrontAng :LREAL := 49.18*2*g_deg2Rad;
	AB :LREAL := 2.8;
	BC:LREAL := 5.26;
	Angle_Initial_A:LREAL := 16.6 * g_deg2Rad; 
	SIN_C,Angle_Initial_C,End_Angle_Single,Angle_Inc_C,Angle_C,SIN_A,Angle_A,Angle_Inc_A:LREAL;
END_VAR

//**************已知：器械前端开合角，求解：末端开合角***************//

//输入合法性判断，物理极限是[16.6*2，49.18*2]度
frontAngle := LIMIT(minFrontAng, frontAngle, maxFrontAng);


SIN_C:=AB*SIN(Angle_Initial_A)/BC;
Angle_Initial_C:=ASIN(SIN_C);

Angle_Inc_A:=frontAngle/2;
Angle_A:=Angle_Initial_A+Angle_Inc_A;

SIN_C:=AB*SIN(Angle_A)/BC;
Angle_C:=ASIN(SIN_C);

Angle_Inc_C:=Angle_C-Angle_Initial_C;
endAngle:=Angle_Inc_C*2;
END_METHOD

METHOD gripperAngleInverseTransform_ID12 : BOOL
VAR_INPUT
	endAngle:LREAL;
END_VAR
VAR_OUTPUT
	frontAngle:LREAL;
	Succeed:BOOL;
END_VAR
VAR
	minEndAng :LREAL  := 0;
	maxEndAng :LREAL := 38*g_deg2Rad;
	AB :LREAL := 2.8;
	BC:LREAL := 5.26;
	Angle_Initial_A:LREAL := 16.6 * g_deg2Rad; 
	
	SIN_C,Angle_Initial_C,End_Angle_Single,Angle_Inc_C,Angle_C,SIN_A,Angle_A,Angle_Inc_A:LREAL;
END_VAR

//***************已知：器械末端开合角，求解：前端开合角********************//

//输入合法性判断，物理极限是[0,30]度
endAngle:= LIMIT(minEndAng, endAngle, maxEndAng);

SIN_C:=AB*SIN(Angle_Initial_A)/BC;
Angle_Initial_C:=ASIN(SIN_C);

End_Angle_Single:=endAngle/2;
Angle_Inc_C:=End_Angle_Single;
Angle_C:=Angle_Initial_C+Angle_Inc_C;

SIN_A:=BC*SIN(Angle_C)/AB;
Angle_A:=ASIN(SIN_A);

Angle_Inc_A:=Angle_A-Angle_Initial_A;
frontAngle:=Angle_Inc_A*2;
END_METHOD

PROPERTY ID : INT
GET
ID:=m_ID;
END_GET
END_PROPERTY

// convert motor joint position to DH joint position
METHOD PUBLIC instruFK : BOOL
VAR_IN_OUT CONSTANT
	// motor joint position of slave arm
	i_jntPos :Vec8d;
END_VAR

VAR_IN_OUT
	// instrument DH  joint positon
	r_DHJntPos :Vec6d;

	// gripper angle
	r_gripAngle :LREAL;
END_VAR

VAR
	jntPosL1,jntPosL2,jntPosL3,jntPosL4,jntPosL5 :LREAL;
	gripAngle:LREAL;
END_VAR
r_DHJntPos[1]:=i_jntPos[1];
r_DHJntPos[2]:=i_jntPos[2];
r_DHJntPos[3]:=i_jntPos[3];


jntPosL1:=i_jntPos[4];
jntPosL2:=i_jntPos[5];
jntPosL3:=i_jntPos[6];
jntPosL4:=i_jntPos[7];
jntPosL5:=i_jntPos[8];
r_DHJntPos[4]:=jntPosL4/m_kinematicParameters.kx;
r_DHJntPos[5]:=jntPosL3/m_kinematicParameters.ky;
r_DHJntPos[6]:=(jntPosL1-jntPosL2-2*r_DHJntPos[5]*m_kinematicParameters.k13*m_kinematicParameters.kz)/(2*m_kinematicParameters.open_direction*m_kinematicParameters.kz);

gripAngle:=(jntPosL1+jntPosL2)/(m_kinematicParameters.open_direction*m_kinematicParameters.kz);
IF (12=m_ID) THEN//细齿无创抓钳
	gripperAngleForwardTransform_ID12(frontAngle:= gripAngle, endAngle=> r_gripAngle);

ELSIF (16 =m_ID) THEN//单级电钩
	r_gripAngle:=0;
	
ELSE
	r_gripAngle:=gripAngle;
END_IF
END_METHOD

METHOD instruIK : BOOL
VAR_INPUT
	// DH  joint positon
	i_jntPosX :LREAL;
	i_jntPosY :LREAL;
	i_jntPosZ :LREAL;
	
	// gripper angle
	i_gripAngle :LREAL;
	
	// joint current
	i_jntCurrentL1 :LREAL;
	i_jntCurrentL2 :LREAL;
END_VAR
VAR_OUTPUT
	angle_slave_L1:lreal;
	angle_slave_L2:lreal;
	angle_slave_L3:lreal;
	angle_slave_L4:lreal;
	angle_slave_L5:lreal;
END_VAR
VAR
	gripAngle:LREAL;
	k1:INT;
	rot_x:lreal;
	rot_y:lreal;
	rot_z:lreal;

	kx,ky,kz,k13,k23:LREAL;
	open_direction:INT;
	
	d,ra:LREAL;
	angle_slave_L1_p1,angle_slave_L1_p2,angle_slave_L1_p3,angle_slave_L1_p4,angle_slave_L3_p1:LREAL;
	angle_slave_L2_p1,angle_slave_L2_p2,angle_slave_L2_p3,angle_slave_L2_p4:LREAL;
	
	wusi_compensate_p1:BOOL;
	wusi_len_to_angle_L1,wusi_len_to_angle_L2:LREAL;
	
	wusi_compensate_p2:BOOL;
	wusi_compensate_p2_first:BOOL:=TRUE;
	rz_first:LREAL;
	case_selected:REAL;
	
	rz_target,rz_actual:LREAL;
	return_direction_limit_positive,return_direction_limit_negative:LREAL;
	angle_rz_before_offset:LREAL;
	
	L1_Current,L2_Current:LREAL;
	L1_Target_Current,L2_Target_Current:LREAL;
	L1_Current_Error,L2_Current_Error:LREAL;
	L1_Velocity,L2_Velocity:LREAL;
	L1_Pos_INC,L2_Pos_INC:LREAL;
	
	//L1_Pos_INC_last,L2_Pos_INC_last:LREAL;
	L1_Pos_INC_sum,L2_Pos_INC_sum:LREAL;
	Pos_INC_sum_max:LREAL:=0.3;
	L3Offset:LREAL:=-3;
END_VAR


//*********************动力盒关节逆向运动学，根据空间关节计算L1-L5**************************//
IF (12=m_ID) THEN//细齿无创抓钳
	gripperAngleInverseTransform_ID12(endAngle:= i_gripAngle, frontAngle=> gripAngle);
	
ELSIF 16 = m_ID THEN//单级电钩\电铲
	gripAngle:=0;
	
ELSE
	gripAngle:=i_gripAngle;
END_IF


//*******************************基本逆向运动学计算***************************************//
//angle_slave_L3:=rot_y*ky;
angle_slave_L4:=rot_x*kx;
angle_slave_L5:=0;
d:=open_direction;

//保证输入的开合角必须大于等于0
IF (gripAngle>=-2) THEN
	ra:=gripAngle;
	//program_control.Gap_Compensation:=TRUE; //打开反向间隙补偿，保证姿态
ELSE
	ra:=-0.0001; //ra:=0;	
	//program_control.Gap_Compensation:=FALSE; //关闭反向间隙补偿，保证夹持力
END_IF

angle_slave_L1_p1:=rot_y*k13*kz+d*rot_z*kz+d*ra*kz/2;
angle_slave_L2_p1:=-rot_y*k23*kz-d*rot_z*kz+d*ra*kz/2;






//******************************器械闭合，是否需要补偿丝的弹性**********************************//
IF (gripAngle<-0.3) THEN
	wusi_compensate_p1:=TRUE;
ELSE
	wusi_compensate_p1:=FALSE;
END_IF

//就目前来说，无法根据器械的夹持力，推算电机扭矩，然后根据电机扭矩计算丝的伸长，此处直接给出丝的伸长量对应的电机角度
IF (wusi_compensate_p1=TRUE) THEN
	wusi_len_to_angle_L1:=0.22; //0.2136
	wusi_len_to_angle_L2:=0.22; //0.2136
	
	//理论数据(值0.2136)暂时有误，以下采用实验数据
	angle_slave_L1_p2:=wusi_len_to_angle;
	angle_slave_L2_p2:=wusi_len_to_angle;
ELSE
	angle_slave_L1_p2:=0;
	angle_slave_L2_p2:=0;
END_IF





//********器械夹紧，并且做偏转运动，因为丝的弹性，造成器械偏转姿态不准确，就需要补偿丝的弹性******//
k1:=m_ID;
IF (wusi_compensate_p1=TRUE) THEN	
	IF (wusi_compensate_p2_first=TRUE) THEN
		wusi_compensate_p2_first:=FALSE;
		rz_first:=rot_z;  //器械初次夹紧，记录此时的偏转角	
	END_IF
	
ELSE
	wusi_compensate_p2_first:=TRUE;
	rz_first:=0;
	surgical_instrument_move_direction_now[k1]:=0;
	surgical_instrument_move_direction_last[k1]:=0;
	surgical_Instrument_Pos_max[k1]:=0;
	surgical_Instrument_Pos_min[k1]:=0;
	
	L1_target_pos_offset[k1]:=0;
	L2_target_pos_offset[k1]:=0;
	L1_actual_pos_offset[k1]:=0;
	L2_actual_pos_offset[k1]:=0;
	
	L1_target_pos_offset_last[k1]:=0;
	L2_target_pos_offset_last[k1]:=0;
	case_selected:=0;	
END_IF





IF (wusi_compensate_p1=TRUE) THEN
	rz_target:=rot_z;
	return_direction_limit_positive:=surgical_instrument_return_direction_limit; 
	return_direction_limit_negative:=-surgical_instrument_return_direction_limit;
	
	
	//初始化器械偏转方向
	IF (surgical_instrument_move_direction_now[k1]=0) THEN
		IF (rz_target-rz_first)>return_direction_limit_positive THEN
			surgical_instrument_move_direction_now[k1]:=1; //将器械偏转方向初始化为正方向
			
		ELSIF (rz_target-rz_first)<return_direction_limit_negative THEN
			surgical_instrument_move_direction_now[k1]:=-1; //将器械偏转方向初始化为负方向
			
		ELSE
			surgical_instrument_move_direction_now[k1]:=0; //器械偏转角还不够大，判定方向没有改变
		END_IF
	END_IF


	//记录系统的极值，且更新运动方向
	angle_rz_before_offset:=rot_z;
	IF (.surgical_instrument_move_direction_last[k1]=0) THEN
		//如果上一时刻还没有运动，且当前正向运动，更新系统最大位置
		IF (surgical_instrument_move_direction_now[k1]=1) THEN
			surgical_Instrument_Pos_max[k1]:=angle_rz_before_offset;
			
		//如果上一时刻还没有运动，且当前负向运动，更新系统最小位置
		ELSIF (surgical_instrument_move_direction_now[k1]=-1) THEN
			surgical_Instrument_Pos_min[k1]:=angle_rz_before_offset;
			
		ELSE
			//如果上一时刻没有运动，当前也没有运动，不用更新系统位置
		END_IF
	END_IF
	
	
	IF (surgical_instrument_move_direction_last[k1]=1) THEN
		//如果上一次运动方向为正，且最新目标位置更大，则更新最大目标位置
		IF (angle_rz_before_offset>surgical_Instrument_Pos_max[k1]) THEN
			surgical_Instrument_Pos_max[k1]:=angle_rz_before_offset;
			
		//如果上一次运动方向为正，且最新位置的目标值反向到一定程度，则确定反向
		ELSIF (angle_rz_before_offset-surgical_Instrument_Pos_max[k1])<return_direction_limit_negative THEN
			surgical_instrument_move_direction_now[k1]:=-1;
			surgical_Instrument_Pos_min[k1]:=angle_rz_before_offset;
			
		ELSE
				//如果上一次运动方向为正，最新位置反向，但是没有到判断极限，则仍认为方向不变
		END_IF
	END_IF


	IF (surgical_instrument_move_direction_last[k1]=-1) THEN
		//如果上一次运动方向为负，且最小目标位置更小，则更新最小目标位置
		IF (angle_rz_before_offset<surgical_Instrument_Pos_min[k1]) THEN
			surgical_Instrument_Pos_min[k1]:=angle_rz_before_offset;
			
		//如果上一次运动方向为负，且最新位置的目标值反向到一定程度，则确定反向
		ELSIF (angle_rz_before_offset-surgical_Instrument_Pos_min[k1])>return_direction_limit_positive THEN
			surgical_instrument_move_direction_now[k1]:=1;
			surgical_Instrument_Pos_max[k1]:=angle_rz_before_offset;
			
		ELSE
				//如果上一次运动方向为负，最新位置反向，但是没有到判断极限，则仍认为方向不变
		END_IF
	END_IF
	
	
	//器械夹紧，并且做偏转运动，因为丝的弹性，造成器械偏转姿态不准确，就需要补偿丝的弹性
	IF (surgical_instrument_move_direction_last[k1]=surgical_instrument_move_direction_now[k1]) THEN
		//如果两次的目标运动方向相同，则目标偏置和实际偏置都保持不变
		L1_target_pos_offset[k1]:=L1_target_pos_offset_last[k1];
		L2_target_pos_offset[k1]:=L2_target_pos_offset_last[k1];
		L3_target_pos_offset[k1]:=L3_target_pos_offset_last[k1];
		
		L1_actual_pos_offset[k1]:=L1_actual_pos_offset_last[k1];
		L2_actual_pos_offset[k1]:=L2_actual_pos_offset_last[k1];
		L3_actual_pos_offset[k1]:=L3_actual_pos_offset_last[k1];
		
		case_selected:=5;
		
	ELSIF (surgical_instrument_move_direction_last[k1]=0) AND (surgical_instrument_move_direction_now[k1]=1) THEN
		//如果上一次为零，现在为正方向  	  L1:目标位置添加负向补偿，实际位置添加正向补偿    L2:目标位置和实际位置不补偿
		L1_target_pos_offset[k1]:=-surgical_instrument_offset[k1];
		L1_actual_pos_offset[k1]:=surgical_instrument_offset[k1];
		
		L2_target_pos_offset[k1]:=0;
		L2_actual_pos_offset[k1]:=0;
		
		
		case_selected:=1;
		
	ELSIF (surgical_instrument_move_direction_last[k1]=0) AND (surgical_instrument_move_direction_now[k1]=-1) THEN
		//如果上一次为零，现在为负方向  	  L1:目标位置和实际位置不补偿    L2:目标位置添加负向补偿，实际位置添加正向补偿
		L1_target_pos_offset[k1]:=0;
		L1_actual_pos_offset[k1]:=0;
		
		L2_target_pos_offset[k1]:=-surgical_instrument_offset[k1];
		L2_actual_pos_offset[k1]:=surgical_instrument_offset[k1];
		
		case_selected:=2;
		
	ELSIF (surgical_instrument_move_direction_last[k1]=1) AND (surgical_instrument_move_direction_now[k1]=-1) THEN
		//如果上一次为正方向，现在为负方向，L1:无需补偿    L2:目标位置添加负向补偿，实际位置添加正向补偿
		L1_target_pos_offset[k1]:=0;
		L1_actual_pos_offset[k1]:=0;
		
		L2_target_pos_offset[k1]:=-surgical_instrument_offset[k1];
		L2_actual_pos_offset[k1]:=surgical_instrument_offset[k1];
		
		
		case_selected:=3;
		
	ELSIF (surgical_instrument_move_direction_last[k1]=-1) AND (surgical_instrument_move_direction_now[k1]=1) THEN
		//如果上一次为负方向，现在为正方向，L1:目标位置添加负向补偿，实际位置添加正向补偿    L2:无需补偿
		L1_target_pos_offset[k1]:=-surgical_instrument_offset[k1];
		L1_actual_pos_offset[k1]:=surgical_instrument_offset[k1];
		
		L2_target_pos_offset[k1]:=0;
		L2_actual_pos_offset[k1]:=0;
		
		
		case_selected:=4;
	END_IF
	
	//参数赋值
	L1_target_pos_offset_last[k1]:=L1_target_pos_offset[k1];
	L2_target_pos_offset_last[k1]:=L2_target_pos_offset[k1];
	L3_target_pos_offset_last[k1]:=L3_target_pos_offset[k1];

	L1_actual_pos_offset_last[k1]:=L1_actual_pos_offset[k1];
	L2_actual_pos_offset_last[k1]:=L2_actual_pos_offset[k1];
	L3_actual_pos_offset_last[k1]:=L3_actual_pos_offset[k1];
	
	
	//夹紧偏摆时造成的俯仰跳动补偿
	L3_target_pos_offset[k1]:=((i_jntCurrentL1-i_jntCurrentL2)/250)*L3Offset*g_deg2Rad;
	L3_actual_pos_offset[k1]:=-((i_jntCurrentL1-i_jntCurrentL2)/250)*L3Offset*g_deg2Rad;

	
	//补偿添加	
	angle_slave_L1_p3:=L1_target_pos_offset[k1];
	angle_slave_L2_p3:=L2_target_pos_offset[k1];
	angle_slave_L3_p1:=L3_target_pos_offset[k1];
	//更新数据
	surgical_instrument_move_direction_last[k1]:=surgical_instrument_move_direction_now[k1];
	
ELSE
	L1_actual_pos_offset[k1]:=0;
	L2_actual_pos_offset[k1]:=0;
	L3_actual_pos_offset[k1]:=0;
	angle_slave_L1_p3:=0;
	angle_slave_L2_p3:=0;
	angle_slave_L3_p1:=0;
END_IF





//*****************第四部分，控制夹持力，根据电流，给定一个由偏差产生的速度********************//
IF (wusi_compensate_p1=TRUE) AND (Robot_clamping_force_control[k1]=TRUE) THEN
	L1_Current:=i_jntCurrentL1;
	L2_Current:=i_jntCurrentL2;
	
	L1_Target_Current:=force_control_target_current;
	L2_Target_Current:=force_control_target_current;
	
	L1_Current_Error:=L1_Target_Current-L1_Current;
	L2_Current_Error:=L2_Target_Current-L2_Current;
	
	L1_Velocity:=force_control_factor_P*L1_Current_Error;
	L2_Velocity:=force_control_factor_P*L2_Current_Error;
	
	L1_Pos_INC:=L1_Velocity*g_slaveArmCtrlCycleTime;
	L2_Pos_INC:=L2_Velocity*g_slaveArmCtrlCycleTime;
	
	L1_Pos_INC_sum:=L1_Pos_INC+L1_Pos_INC_sum;
	L2_Pos_INC_sum:=L2_Pos_INC+L2_Pos_INC_sum;
	
	IF (L1_Pos_INC_sum>Pos_INC_sum_max) THEN
		L1_Pos_INC_sum:=Pos_INC_sum_max;
	ELSIF (L1_Pos_INC_sum<-Pos_INC_sum_max) THEN
		L1_Pos_INC_sum:=-Pos_INC_sum_max;
	END_IF
	
	IF (L2_Pos_INC_sum>Pos_INC_sum_max) THEN
		L2_Pos_INC_sum:=Pos_INC_sum_max;
	ELSIF (L2_Pos_INC_sum<-Pos_INC_sum_max) THEN
		L2_Pos_INC_sum:=-Pos_INC_sum_max;
	END_IF	
	
	//angle_slave_L1_p4:=L1_Pos_INC_sum;
	//angle_slave_L2_p4:=L2_Pos_INC_sum;
	angle_slave_L1_p4:=0.3;
	angle_slave_L2_p4:=0.3;
	
ELSE
	angle_slave_L1_p4:=0;
	angle_slave_L2_p4:=0;
	L1_Pos_INC_sum:=0;
	L2_Pos_INC_sum:=0;
END_IF


angle_slave_L1:=angle_slave_L1_p1;//+angle_slave_L1_p3;//+angle_slave_L1_p4;
angle_slave_L2:=angle_slave_L2_p1;//+angle_slave_L2_p3;//+angle_slave_L2_p4;
//angle_slave_L3:=angle_slave_L3_p1;
angle_slave_L3:=rot_y*ky+angle_slave_L3_p1;
//ngle_slave_L1:=angle_slave_L1_p1+angle_slave_L1_p2+angle_slave_L1_p3;//+angle_slave_L1_p4;
//angle_slave_L2:=angle_slave_L2_p1+angle_slave_L2_p2+angle_slave_L2_p3;//+angle_slave_L2_p4;
END_METHOD

PROPERTY instruType : E_InstrumentType
GET
instruType:=m_type;
END_GET
END_PROPERTY

PROPERTY kinematicParameters :REFERENCE TO ST_InstruParameters
GET
kinematicParameters ref=m_kinematicParameters;
END_GET
END_PROPERTY

PROPERTY maxUsageCounts : INT
GET
maxUsageCounts:=m_maxUsageCounts;
END_GET
END_PROPERTY

METHOD readParameters : BOOL
VAR_INPUT
END_VAR
// TODO: read m_kinematic parameters from chip
END_METHOD

METHOD reset : BOOL
VAR_INPUT
END_VAR
m_ID := 0;
m_seriesNum :=0;
m_type :=InstruType_UNKNOWM;
END_METHOD

PROPERTY SeriesNum : ULINT
GET
SeriesNum:=m_seriesNum;
END_GET
END_PROPERTY

PROPERTY usageCounts : INT
GET
usageCounts:=m_usageCounts;
END_GET
END_PROPERTY

END_FUNCTION_BLOCK

// ---- AgiMaths/MatrixLib/invMat6.TcPOU
FUNCTION invMat6 : bool
VAR_IN_OUT CONSTANT
	mat :Mat6d;
END_VAR
VAR_IN_OUT
	invMat : Mat6d;
END_VAR
VAR
	n:INT:=6;
	m:INT:=1;
	b :ARRAY[1..6] OF LREAL := [6(0)];
	indxc,indxr, ipiv:ARRAY[1..6] OF INT := [6(0)];

	
	i,icol, irow, j,k,l,ll: INT;
	big, dum, pivinv,tmp: LREAL;
END_VAR

invMat := mat;
FOR i:=1 TO n DO   
    big:=0.0;
    FOR j:=1 TO n DO  
        IF (ipiv[j] <> 1) THEN
            FOR k:=1 TO n DO 
                IF (ipiv[k] = 0) THEN
                    IF (ABS(invMat[j,k]) >= big) THEN
                        big:=ABS(invMat[j,k]);
                        irow:=j;
                        icol:=k;
                    END_IF
                END_IF
            END_FOR
        END_IF
    END_FOR
    ipiv[icol]:=ipiv[icol]+1;
    
    IF (irow <> icol) THEN
        FOR l:=1 TO n DO 
            tmp:=invMat[irow,l];
            invMat[irow,l]:=invMat[icol,l];
            invMat[icol,l]:=tmp;
        END_FOR
 (*       FOR  l:=1 TO m DO  
            tmp:=b[irow,l];
            b[irow,l]:=b[icol,l];
            b[icol,l]:=tmp;
        END_FOR*)
    END_IF
	
    indxr[i]:=irow; 
    indxc[i]:=icol;
	
    IF ABS(invMat[icol,icol]) < g_smallNum THEN 
          invMat6:=FALSE;
		  RETURN;
    END_IF
	
    pivinv:=1.0/invMat[icol,icol];
    invMat[icol,icol]:=1.0;
    FOR l:=1 TO n DO  
        invMat[icol,l] := invMat[icol,l]*pivinv;
    END_FOR
 (*   FOR l:=1 TO m DO 
        b[icol,l] := b[icol,l]*pivinv;
    END_FOR*)
    FOR ll:=1 TO n DO  
        IF (ll <> icol) THEN 
            dum:=invMat[ll,icol];
            invMat[ll,icol]:=0.0;
            FOR l:=1 TO n DO  
                invMat[ll,l]:=invMat[ll,l] - invMat[icol,l]*dum;
            END_FOR
   (*         FOR l:=1 TO m DO  
                b[ll,l]:=b[ll,l] - b[icol,l]*dum;
            END_FOR*)
        END_IF
    END_FOR

END_FOR


FOR l:=n-1 TO 1 BY -1 DO 
    IF (indxr[l] <> indxc[l]) THEN
        FOR k:=1 TO n DO
            tmp:=invMat[k,indxr[l]];
            invMat[k,indxr[l]]:=invMat[k,indxc[l]];
            invMat[k,indxc[l]]:=tmp;
        END_FOR
    END_IF
END_FOR

invMat6:=TRUE;

END_FUNCTION

// ---- FBs_SlaveControllers/FB_SlaveCtrlSelfCheck.TcPOU
// Brief: Slave Arm Run Self-check Trajectory
FUNCTION_BLOCK PUBLIC FB_SlaveCtrlSelfCheck EXTENDS FB_SlaveArmCtrlBase
VAR_INPUT
END_VAR
VAR_OUTPUT
END_VAR
VAR
	m_selfCheckTrajIdx: INT := 1;
	m_slefCheckPlanner: ARRAY[1..GVL_SlaveControlParameters.g_selfCheckMotionNum] OF FB_TrajMoveJ;
	
END_VAR

// override this function in each exact controller
METHOD PROTECTED calcCmdJntPos : BOOL
VAR_INPUT
	motionScale :LREAL;
	masterIdx :INT;
END_VAR

VAR_IN_OUT CONSTANT
	i_slaveArm :FB_SlaveArm;
	i_masterStatus :ST_MasterStatus;
END_VAR

VAR 
	i :INT;
	curJntVel :Vec8d;
END_VAR
// check if planner is ready
IF m_slefCheckPlanner[m_selfCheckTrajIdx].isGene = FALSE THEN
	calcCmdJntPos:=FALSE;
	RETURN;
END_IF

// traj plan
calcCmdJntPos :=m_slefCheckPlanner[m_selfCheckTrajIdx].evaluate(m_timePeriod, jntPos=> m_cmdJntPos, jntVel=>m_cmdJntVel, jntAcc=> m_cmdJntAcc);

// check if to transit to next segment
curJntVel :=i_slaveArm.curJntVel;
IF(m_timePeriod > m_slefCheckPlanner[m_selfCheckTrajIdx].duration  AND vecNorm(curJntVel)<7*GVL_SlaveControlParameters.g_jntStaticVelThres) THEN
	m_selfCheckTrajIdx:=m_selfCheckTrajIdx+1;
	m_timePeriod:=0;
END_IF

// check if to terminated
IF(m_selfCheckTrajIdx > GVL_SlaveControlParameters.g_selfCheckMotionNum) THEN
	m_isFinished:=TRUE;
END_IF
END_METHOD

METHOD PUBLIC init : BOOL
VAR_IN_OUT CONSTANT
	i_slaveArm	:FB_SlaveArm;
END_VAR
VAR_IN_OUT 
	r_slaveArmCtrlCmd :ST_SlaveArmCtrlCmds;
END_VAR

VAR
	i,j :INT;
	startJntPos,endJntPos :Vec8d;
END_VAR
SUPER^.Init(i_slaveArm,r_slaveArmCtrlCmd);
m_selfCheckTrajIdx :=1;

// traj plan
// fisrt segment
startJntPos:=i_slaveArm.curJntPos;
FOR j:=1 TO 7 DO 
endJntPos[j]:=GVL_SlaveControlParameters.g_selfCheckPosture[1,j];
END_FOR
m_slefCheckPlanner[1].init(startJntPos,endJntPos,GVL_SlaveControlParameters.g_selfCheckMaxjntVel,
					GVL_SlaveControlParameters.g_selfCheckMaxjntAcc,GVL_SlaveControlParameters.g_selfCheckMaxjntJerk);
// other segments
FOR i:=2 TO GVL_SlaveControlParameters.g_selfCheckMotionNum DO 
	FOR j:=1 TO 7 DO 
		startJntPos[j]:=GVL_SlaveControlParameters.g_selfCheckPosture[i-1,j];
		endJntPos[j]:=GVL_SlaveControlParameters.g_selfCheckPosture[i,j];
	END_FOR
	m_slefCheckPlanner[i].init(startJntPos,endJntPos,GVL_SlaveControlParameters.g_selfCheckMaxjntVel,
						GVL_SlaveControlParameters.g_selfCheckMaxjntAcc,GVL_SlaveControlParameters.g_selfCheckMaxjntJerk);
END_FOR
END_METHOD

END_FUNCTION_BLOCK

// ---- FBs_SlaveControllers/FB_SlaveArmCtrlBase.TcPOU
// Slave Arm Base Controller, Hold at Current Posture
FUNCTION_BLOCK FB_SlaveArmCtrlBase IMPLEMENTS I_SlaveArmCtrl
VAR_INPUT
END_VAR
VAR_OUTPUT
END_VAR
VAR
	// flag if the controller has finished all its jobs
	m_isFinished:BOOL:=FALSE;
	
	// controller execute time period
	m_timePeriod :LREAL:=0;
	
	// arm control data
	m_cmdJntPos : VEC8d;
	m_cmdJntVel : VEC8d;
	m_cmdJntAcc : VEC8d;
	m_cmdJntTrq : VEC8d;
	m_jntOPMode : Vec8i;
	m_jntEnableFlag :Vec8i;
	m_cmdCartPose : ST_Frame;
	m_cmdCartTwist : Vec6d;
END_VAR

// override this function in each exact controller
METHOD PROTECTED calcCmdJntPos : BOOL
VAR_INPUT
	motionScale :LREAL;
	masterIdx :INT;
END_VAR

VAR_IN_OUT CONSTANT
	i_slaveArm :FB_SlaveArm;
	i_masterStatus :ST_MasterStatus;
END_VAR
END_METHOD

// override this function in each exact controller
METHOD PROTECTED calcCmdJntTrq : BOOL
VAR_INPUT
	motionScale :LREAL;
	masterIdx :INT;
END_VAR

VAR_IN_OUT CONSTANT
	i_slaveArm :FB_SlaveArm;
	i_masterStatus :ST_MasterStatus;
END_VAR
// set joint torque to zero in default
m_cmdJntTrq := g_zeroVec8d;
END_METHOD

METHOD checkToHoldLastCmds : BOOL
VAR_IN_OUT CONSTANT
	i_slaveArm :FB_SlaveArm;
	i_slaveArmCtrlCmd :ST_SlaveArmCtrlCmds;
END_VAR
VAR
	j:INT;
	maxJntErr:LREAL;
	jntCtrlErr:Vec7d;
END_VAR
// check if to hold the command joint position unchanged
vecSub(i_slaveArmCtrlCmd.m_cmdJntPos, i_slaveArm.m_curJntPos,jntCtrlErr);
maxJntErr:=0.0;
FOR j:=1 TO g_sJntNum DO
	maxJntErr:= MAX(maxJntErr, ABS(jntCtrlErr[j]));
END_FOR

IF maxJntErr<GVL_SlaveControlParameters.g_jntCtrlErrForCmdHold THEN
	m_cmdJntPos:=i_slaveArmCtrlCmd.m_cmdJntPos;
ELSE
	m_cmdJntPos:=i_slaveArm.curJntPos;
END_IF
END_METHOD

// override this function in each exact controller
// NOTICE: set joint control mode here, and do some initialization if needed
METHOD PUBLIC init : BOOL
VAR_IN_OUT CONSTANT
	i_slaveArm	:FB_SlaveArm;
END_VAR
VAR_IN_OUT 
	r_slaveArmCtrlCmd :ST_SlaveArmCtrlCmds;
END_VAR
m_timePeriod:=0;
m_jntEnableFlag :=g_onesVec8i;
m_jntEnableFlag[8]:=0; // L5 joint on instrument power box is unused currently 
m_jntOPMode:=g_slaveAllPosMode;
m_cmdCartPose:=i_slaveArm.curCartPose;
m_cmdCartTwist:=g_zeroVec6d;
m_cmdJntPos:=i_slaveArm.curJntPos;
m_cmdJntVel:=g_zeroVec8d;
m_cmdJntAcc:=g_zeroVec8d;
m_cmdJntTrq:=g_zeroVec8d;

// update commands to arm
r_slaveArmCtrlCmd.m_jntEnableFlag :=m_jntEnableFlag;
r_slaveArmCtrlCmd.m_cmdCartPose:=m_cmdCartPose;
r_slaveArmCtrlCmd.m_cmdCartTwist:=m_cmdCartTwist;
r_slaveArmCtrlCmd.m_cmdJntPos:=m_cmdJntPos;
r_slaveArmCtrlCmd.m_cmdJntVel:=m_cmdJntVel;
r_slaveArmCtrlCmd.m_cmdJntAcc:=m_cmdJntAcc;
r_slaveArmCtrlCmd.m_cmdJntTrq:=m_cmdJntTrq;
r_slaveArmCtrlCmd.m_jntOPMode:=m_jntOPMode;
END_METHOD

PROPERTY isFinished : BOOL
GET
isFinished:=m_isFinished;
END_GET
END_PROPERTY

{warning '添加方法实现'}
METHOD reset : BOOL
m_isFinished:=FALSE;
m_timePeriod:=0;
END_METHOD

{warning '添加方法实现'}
METHOD run : BOOL
VAR_INPUT
	motionScale :LREAL;
	masterIdx :INT;
END_VAR

VAR_IN_OUT CONSTANT
	i_slaveArm :FB_SlaveArm;
	i_masterStatus :ST_MasterStatus;
END_VAR
VAR_IN_OUT
	r_slaveArmCtrlCmd :ST_SlaveArmCtrlCmds;
END_VAR
VAR
	i:INT;
END_VAR
IF m_isFinished THEN
	RETURN;
END_IF

// check if arm enabled
IF FALSE = i_slaveArm.isEnabled(m_jntEnableFlag) THEN
//	RETURN;
END_IF

// calculate command joint position--Motion control
calcCmdJntPos(motionScale, masterIdx, i_slaveArm,i_masterStatus);

// calculate command joint torque -- Force control
calcCmdJntTrq(motionScale, masterIdx, i_slaveArm,i_masterStatus);

// update commands to arm
r_slaveArmCtrlCmd.m_jntEnableFlag :=m_jntEnableFlag;
r_slaveArmCtrlCmd.m_cmdCartPose:=m_cmdCartPose;
r_slaveArmCtrlCmd.m_cmdCartTwist:=m_cmdCartTwist;
r_slaveArmCtrlCmd.m_cmdJntPos:=m_cmdJntPos;
r_slaveArmCtrlCmd.m_cmdJntVel:=m_cmdJntVel;
r_slaveArmCtrlCmd.m_cmdJntAcc:=m_cmdJntAcc;
r_slaveArmCtrlCmd.m_cmdJntTrq:=m_cmdJntTrq;
r_slaveArmCtrlCmd.m_jntOPMode:=m_jntOPMode;

// update time period
m_timePeriod := m_timePeriod+g_slaveArmCtrlCycleTime;
END_METHOD

END_FUNCTION_BLOCK

// ---- FBs_TrajectoryPlanning/FB_TrajMoveJ.TcPOU
FUNCTION_BLOCK FB_TrajMoveJ EXTENDS FB_TrajBase
VAR_OUTPUT
END_VAR
VAR
	// move vector in joint space
	m_startPos:Vec8d;
	m_targetPos:Vec8d;
	m_moveDir : Vec8d;
	m_moveDistance :LREAL;
	
	// doubleS planning for move distance
	m_doubleS :FB_BasicDoubleS;
END_VAR

METHOD evaluate : BOOL
VAR_INPUT
	t :LREAL;
END_VAR

VAR_OUTPUT
	jntPos,jntVel, jntAcc :vec8d;
END_VAR
VAR
	q,q_dot,q_ddot :LREAL;
	moveRange :Vec8d;
END_VAR
evaluate:=m_doubleS.evaluate(t,q=>q,q_dot=>q_dot, q_ddot=>q_dot);
IF evaluate =FALSE THEN
	RETURN;
END_IF

vecMultiNum(m_moveDir,q, moveRange);
vecAdd(moveRange, m_startPos,jntPos);
vecMultiNum(m_moveDir,q_dot, jntVel);
vecMultiNum( m_moveDir,q_ddot, jntAcc);
END_METHOD

METHOD init : BOOL
VAR_INPUT
	i_startJntPos :Vec8d;
	i_targetJntPos :Vec8d;
	i_maxJntVel : Vec8d;
	i_maxJntAcc : Vec8d;
	i_maxJntJerk :Vec8d;
END_VAR
VAR 
	i:INT;
	maxV, maxA, maxJ :LREAL;
	q:ARRAY[1..2] OF LREAL;
	v:ARRAY[1..2] OF LREAL;
END_VAR
m_startPos:=i_startJntPos;
m_targetPos:=i_targetJntPos;
vecSub(i_targetJntPos, i_startJntPos, m_moveDir);
m_moveDistance := vecNorm(m_moveDir);

IF(m_moveDistance<g_smallNum) THEN
	vecMultiNum(g_onesVec7d,1/8, m_moveDir);;
ELSE
	vecMultiNum( m_moveDir,1/m_moveDistance, m_moveDir);
END_IF

// determian max vel/acc/jerk
maxV:=g_largeNum;
maxA:=g_largeNum;
maxJ:=g_largeNum;
FOR i :=1 TO 7 DO 
	IF ABS(m_moveDir[i])>g_smallNum THEN
		maxV := MIN (maxV, ABS(i_maxJntVel[i]/m_moveDir[i]));
		maxA := MIN (maxA, ABS(i_maxJntAcc[i]/m_moveDir[i]));
		maxJ := MIN (maxJ, ABS(i_maxJntJerk[i]/m_moveDir[i]));
	END_IF
END_FOR

// planning for moving distance
q[1]:=0;
q[2]:=m_moveDistance;
v[1]:=0;
v[2]:=0;
m_doubleS.init(q,v, maxV, maxA, maxJ);
m_duration:=m_doubleS.duration;
m_isGenerated:=m_doubleS.isGene;
END_METHOD

END_FUNCTION_BLOCK

// ---- FBs_SlaveControllers/FB_SlaveCtrlStandBy.TcPOU
// Brief: Slave Arm Standby
FUNCTION_BLOCK PUBLIC FB_SlaveCtrlStandBy EXTENDS FB_SlaveArmCtrlBase
VAR_INPUT
END_VAR
VAR_OUTPUT
END_VAR
VAR
END_VAR

METHOD PUBLIC init : BOOL
VAR_IN_OUT CONSTANT
	i_slaveArm	:FB_SlaveArm;
END_VAR
VAR_IN_OUT 
	r_slaveArmCtrlCmd :ST_SlaveArmCtrlCmds;
END_VAR
SUPER^.Init(i_slaveArm,r_slaveArmCtrlCmd);

// check if to hold the command joint position unchanged
checkToHoldLastCmds(i_slaveArm,r_slaveArmCtrlCmd);
END_METHOD

END_FUNCTION_BLOCK

// ---- FBs_SlaveControllers/FB_SlaveCtrlMountPanel.TcPOU
// Brief: Mounting Panel
FUNCTION_BLOCK PUBLIC FB_SlaveCtrlMountPanel EXTENDS FB_SlaveArmCtrlBase
VAR_INPUT
END_VAR
VAR_OUTPUT
END_VAR
VAR
	// mount status
	m_mountStatus :INT := 0;
	
	// flag if joint is mounted
	m_jointMounted :ARRAY[1..5] OF BOOL := [5(FALSE)];
	
	// mount motion planning
	m_jntOTG :ARRAY[1..5] OF FB_secOrdTrajFilter;
	m_panelMountVel :LREAL := 90* g_deg2Rad;
	m_panelMountAcc :LREAL := PI;
	
	// joint current threshold which indicate motor is buckled with panel
	m_maxJntCurrent :INT := 100;
	
	// command mount motion
	m_mountStepPos :LREAL := 45.0 * g_deg2Rad;
	m_targetMountPos :Vec5d;
END_VAR

// override this function in each exact controller
METHOD PROTECTED calcCmdJntPos : BOOL
VAR_INPUT
	motionScale :LREAL;
	masterIdx :INT;
END_VAR

VAR_IN_OUT CONSTANT
	i_slaveArm :FB_SlaveArm;
	i_masterStatus :ST_MasterStatus;
END_VAR

VAR 
	i :INT;
	curJntPos :Vec8d;
	jntPosErr :Vec8d;
	cycleNum :INT;
END_VAR

curJntPos := i_slaveArm.curJntPos;

CASE m_mountStatus OF
	// To lock joint with panel
	0:
		FOR i:=1 TO 5 DO
			// check joint buckled with panel
			IF ABS(i_slaveArm.filtJntCurrent[i+3])> m_maxJntCurrent THEN 
				m_jointMounted[i]:=TRUE;
				m_targetMountPos[i]:=curJntPos[i+3];
			END_IF
			
			// set command joint position step
			IF FALSE = m_jointMounted[i] THEN
				m_targetMountPos[i]:=curJntPos[i+3]+m_mountStepPos;
			END_IF
		END_FOR
		
		IF (m_jointMounted[1] AND m_jointMounted[2] AND m_jointMounted[3] AND m_jointMounted[4] AND m_jointMounted[5]) or m_timePeriod > 8.0 THEN
			m_mountStatus:=1;
		END_IF
	
	// determine zero position
	1:
		FOR i:=1 TO 5 DO
			cycleNum := LREAL_TO_INT(curJntPos[i+3]/g_2pi);
			IF curJntPos[i+3]> cycleNum* g_2Pi THEN
				m_targetMountPos[i]:=cycleNum* g_2Pi;
			ELSE
				m_targetMountPos[i]:=(cycleNum-1)* g_2Pi;
			END_IF	
		END_FOR
		m_mountStatus :=2;
	
	// move back to zero position
	2:
		m_isFinished:=TRUE;
		FOR i:=1 TO 5 DO
			IF ABS(m_targetMountPos[i]-curJntPos[i+3])>GVL_SlaveControlParameters.g_jntCtrlPosTol THEN
				m_isFinished:=FALSE;
				EXIT;
			END_IF
		END_FOR
END_CASE

// traj plan
FOR i:=1 TO 5 DO
	m_jntOTG[i].run(m_targetMountPos[i],0.0, o_cmdAcc=>m_cmdJntAcc[3+i],o_cmdVel=>m_cmdJntVel[3+i],o_cmdPos=>m_cmdJntPos[i+3]);
END_FOR
END_METHOD

METHOD PUBLIC init : BOOL
VAR_IN_OUT CONSTANT
	i_slaveArm	:FB_SlaveArm;
END_VAR
VAR_IN_OUT 
	r_slaveArmCtrlCmd :ST_SlaveArmCtrlCmds;
END_VAR
VAR
	i : INT;
END_VAR
SUPER^.Init(i_slaveArm,r_slaveArmCtrlCmd);

m_mountStatus:=0;
FOR i:=1 TO 5 DO
	m_targetMountPos[i]:=m_cmdJntPos[i+3];
	m_jntOTG[i].init(m_targetMountPos[i], 0,m_panelMountVel, m_panelMountAcc, g_slaveArmCtrlCycleTime);
	m_jointMounted[i]:=FALSE;
END_FOR
END_METHOD

END_FUNCTION_BLOCK

// ---- FBs_SlaveControllers/FB_SlaveCtrlMountInstru.TcPOU
// Brief: Mounting Instrument
FUNCTION_BLOCK PUBLIC FB_SlaveCtrlMountInstru EXTENDS FB_SlaveArmCtrlBase
VAR_INPUT
END_VAR
VAR_OUTPUT
END_VAR
VAR
	// mount status
	m_mountStatus :INT := 0;
	m_J4mountStatus :INT := 0;
	
	// flag if joint is mounted
	m_jointMounted :ARRAY[1..5] OF BOOL := [5(FALSE)];
	
	// instrument mount motion range
	m_mountMotionAng :Vec5d :=[2*PI, 2*PI, 2*PI, 2*PI, 2*PI];
	
	// instrument mount direction
	m_mountDir :Vec5i :=[1, 1, 1, 1, 1];
	
	// mount motion planning
	m_jntOTG :ARRAY[1..5] OF FB_secOrdTrajFilter;
	m_instruMountVel :LREAL := 2*PI;//30* g_deg2Rad;
	m_instruMountAcc :LREAL := 2*PI;
	
	// track error threshold which indicate motor is buckled with panel
	m_maxTrackErr :LREAL := 5*g_deg2Rad;
	
	//powerbox motor stop vel
	m_stopVel :LREAL := 1*g_deg2Rad;
	
	//Joint 4 rotation angle
	rotAngleJ4 :LREAL := 323*g_deg2Rad;
	
	// joint current threshold which indicate panel is buckled with instrument
	m_maxJntCurrent :INT := 180;
	
	// command mount motion
	m_targetMountPos :Vec8d;
	
	// instrument zero position
	m_instruZeroDeviation :Mat45;
	m_PowerboxZeroPos :Mat45:=[5.75,5.75,5.75-pi,2,   5.75,5.75,5.75-pi,2,   5.75,5.75,5.75-pi,2,   5.75,5.75,5.75-pi,2];
	m_instruZeroDeviationJ4:LREAL;
	
	//instrument clamping Error
	m_Error:BOOL;
	m_ErrorID:DINT;
END_VAR

// override this function in each exact controller
METHOD PROTECTED calcCmdJntPos : BOOL
VAR_INPUT
	motionScale :LREAL;
	masterIdx :INT;
END_VAR

VAR_IN_OUT CONSTANT
	i_slaveArm :FB_SlaveArm;
	i_masterStatus :ST_MasterStatus;
END_VAR

VAR 
	i :INT;
	curJntVel :Vec8d;
	curJntPos :Vec8d;
	jntPosErr :Vec8d;
END_VAR

curJntPos := i_slaveArm.curJntPos;

CASE m_mountStatus OF
	// To lock panel with instrument
	0:
		FOR i:=1 TO 5 DO
			m_ratedCur[i+3]:=200;
			// check joint buckled with instrument
			IF ABS(i_slaveArm.filtJntCurrent[i+3])> m_maxJntCurrent THEN 
				m_jointMounted[i]:=TRUE;
				m_targetMountPos[i+3]:=curJntPos[i+3];
			END_IF
			
			// set target joint position
			IF FALSE = m_jointMounted[i] THEN
				m_targetMountPos[i+3]:=curJntPos[i+3]-m_mountMotionAng[i];
			END_IF
		END_FOR
		
		IF (m_jointMounted[1] AND m_jointMounted[2] AND m_jointMounted[3] AND m_jointMounted[4] AND m_jointMounted[5])  THEN
			IF i_slaveArm.instrument.InstruReadPara.m_InstruReadSucceed THEN//Check whether the data is read successfully
				m_mountStatus:=1;
			ELSE
				m_Error:=TRUE;
				m_ErrorID:=1;
			END_IF
		END_IF
	
	1:// The calculation deviates from the instrument zero position
		(*IF m_instruZeroDeviationJ4>PI THEN //J4
			m_instruZeroDeviation[1,4]:=m_instruZeroDeviationJ4;
		ELSE
			m_instruZeroDeviation[1,4]:=-m_instruZeroDeviationJ4;
		END_IF*)
		m_instruZeroDeviation[1,4]:=rotAngleJ4;
		
		FOR i:=1 TO 3 DO//J1-3
			m_instruZeroDeviation[1,i] := m_PowerboxZeroPos[1,i] - i_slaveArm.linkSingle[i+3] - i_slaveArm.instrument.InstruReadPara.m_InstruPos[1,i];
			IF m_instruZeroDeviation[1,i]>pi THEN
				m_instruZeroDeviation[1,i] := m_instruZeroDeviation[1,i] - 2*PI;
			ELSIF m_instruZeroDeviation[1,i]<-pi THEN
				m_instruZeroDeviation[1,i] := m_instruZeroDeviation[1,i] + 2*PI;
			END_IF
		END_FOR
		m_mountStatus :=2;
	
	
	2:// move back to zero position
	
		// set target joint position
		FOR i:=1 TO 4 DO
			m_targetMountPos[i+3]:=curJntPos[i+3] + m_instruZeroDeviation[1,i];
		END_FOR
		m_mountStatus :=3;
		
		
	3:
		m_isFinished:=TRUE;
		FOR i:=1 TO 5 DO
			IF ABS(m_targetMountPos[i+3]-curJntPos[i+3])>0.05 THEN
				m_isFinished:=FALSE;
				EXIT;
			END_IF
		END_FOR
		
		(*vecSub(m_targetMountPos,curJntPos,jntPosErr);
		IF vecNorm(jntPosErr)<GVL_SlaveControlParameters.g_jntCtrlPosTol THEN
			m_isFinished:=TRUE;
		END_IF*)
		
		(*IF  ABS(m_cmdJntPos[7]-m_targetMountPos[7])< GVL_SlaveControlParameters.g_jntCtrlPosTol THEN 
			m_targetMountPos[7]:=curJntPos[7];
		ELSIF ABS(m_cmdJntPos[7]-m_targetMountPos[7])> GVL_SlaveControlParameters.g_jntCtrlPosTol AND ABS(i_slaveArm.filtJntCurrent[7])> 80 AND i_slaveArm.curJntVel[7]<m_stopVel THEN
			
			m_targetMountPos[i+3]:=curJntPos[7]-rotAngleJ4;//direction of current
			m_mountStatus :=4;
		END_IF*)
		
	4:
		vecSub(m_targetMountPos,curJntPos,jntPosErr);
		IF vecNorm(jntPosErr)<GVL_SlaveControlParameters.g_jntCtrlPosTol THEN
			m_isFinished:=TRUE;
		END_IF
		
END_CASE

